LIN {X 0,Y 190.338,Z 370.744,A -85,B 0,C 180,E1 -22072.2,E2 -22072.2} C_VEL
LIN {X 0,Y 193.251,Z 362.35,A -85,B 0,C 180,E1 -22075.296,E2 -22075.296} C_VEL
LIN {X 0,Y 196.197,Z 353.832,A -85,B 0,C 180,E1 -22077.752,E2 -22077.752} C_VEL
LIN {X 0,Y 199.587,Z 343.318,A -85,B 0,C 180,E1 -22080.116,E2 -22080.116} C_VEL
LIN {X 0,Y 202.903,Z 331.483,A -85,B 0,C 180,E1 -22082.176,E2 -22082.176} C_VEL
LIN {X 0,Y 205.757,Z 319.558,A -85,B 0,C 180,E1 -22083.712,E2 -22083.712} C_VEL
LIN {X 0,Y 208.119,Z 307.146,A -85,B 0,C 180,E1 -22084.886,E2 -22084.886} C_VEL
LIN {X 0,Y 209.878,Z 294.163,A -85,B 0,C 180,E1 -22085.737,E2 -22085.737} C_VEL
LIN {X 0,Y 210.855,Z 279.203,A -85,B 0,C 180,E1 -22086.333,E2 -22086.333} C_VEL
LIN {X 0,Y 212.644,Z 242.014,A -85,B 0,C 180,E1 -22087.513,E2 -22087.513} C_VEL
LIN {X 0,Y 211,Z 228.178,A -85,B 0,C 180,E1 -22088.437,E2 -22088.437} C_VEL
LIN {X 0,Y 205.351,Z 214.211,A -85,B 0,C 180,E1 -22090.309,E2 -22090.309} C_VEL
LIN {X 0,Y 199.119,Z 201.239,A -85,B 0,C 180,E1 -22092.447,E2 -22092.447} C_VEL
LIN {X 0,Y 194.454,Z 192.885,A -85,B 0,C 180,E1 -22094.123,E2 -22094.123} C_VEL
LIN {X 0,Y 191.867,Z 188.463,A -85,B 0,C 180,E1 -22095.097,E2 -22095.097} C_VEL
LIN {X 0,Y 189.584,Z 184.486,A -85,B 0,C 180,E1 -22095.998,E2 -22095.998} C_VEL
LIN {X 0,Y 186.826,Z 180.02,A -85,B 0,C 180,E1 -22097.117,E2 -22097.117} C_VEL
LIN {X 0,Y 186.602,Z 179.438,A -85,B 0,C 180,E1 -22097.318,E2 -22097.318} C_VEL
LIN {X 0,Y 185.459,Z 175.379,A -85,B 0,C 180,E1 -22100.247,E2 -22100.247} C_VEL
LIN {X 0,Y 185.496,Z 175.37,A -85,B 0,C 180,E1 -22102.713,E2 -22102.713} C_VEL
LIN {X 0,Y 185.525,Z 175.365,A -85,B 0,C 180,E1 -22107.971,E2 -22107.971} C_VEL
LIN {X 0,Y 185.542,Z 175.361,A -85,B 0,C 180,E1 -22110.595,E2 -22110.595} C_VEL
LIN {X 0,Y 185.557,Z 175.366,A -85,B 0,C 180,E1 -22115.378,E2 -22115.378} C_VEL
LIN {X 0,Y 185.619,Z 175.361,A -85,B 0,C 180,E1 -22121.178,E2 -22121.178} C_VEL
LIN {X 0,Y 185.691,Z 175.355,A -85,B 0,C 180,E1 -22126.874,E2 -22126.874} C_VEL
LIN {X 0,Y 185.962,Z 175.306,A -85,B 0,C 180,E1 -22131.305,E2 -22131.305} C_VEL
LIN {X 0,Y 186.164,Z 175.274,A -85,B 0,C 180,E1 -22137.837,E2 -22137.837} C_VEL
LIN {X 0,Y 186.371,Z 175.265,A -85,B 0,C 180,E1 -22140,E2 -22140} C_VEL
LIN {X 0,Y 185.875,Z 175.31,A -85,B 0,C 180,E1 -22144.337,E2 -22144.337} C_VEL
LIN {X 0,Y 185.968,Z 175.32,A -85,B 0,C 180,E1 -22148.695,E2 -22148.695} C_VEL
LIN {X 0,Y 185.679,Z 175.336,A -85,B 0,C 180,E1 -22153.127,E2 -22153.127} C_VEL
LIN {X 0,Y 185.619,Z 175.347,A -85,B 0,C 180,E1 -22158.822,E2 -22158.822} C_VEL
LIN {X 0,Y 185.572,Z 175.359,A -85,B 0,C 180,E1 -22164.647,E2 -22164.647} C_VEL
LIN {X 0,Y 185.539,Z 175.372,A -85,B 0,C 180,E1 -22169.5,E2 -22169.5} C_VEL
LIN {X 0,Y 185.492,Z 175.38,A -85,B 0,C 180,E1 -22174.634,E2 -22174.634} C_VEL
LIN {X 0,Y 185.495,Z 175.377,A -85,B 0,C 180,E1 -22177.316,E2 -22177.316} C_VEL
LIN {X 0,Y 185.432,Z 175.385,A -85,B 0,C 180,E1 -22182.703,E2 -22182.703} C_VEL
LIN {X 0,Y 186.407,Z 178.185,A -85,B 0,C 180,E1 -22183.202,E2 -22183.202} C_VEL
LIN {X 0,Y 188.839,Z 180.945,A -85,B 0,C 180,E1 -22184.138,E2 -22184.138} C_VEL
LIN {X 0,Y 191.097,Z 184.353,A -85,B 0,C 180,E1 -22185.017,E2 -22185.017} C_VEL
LIN {X 0,Y 197.59,Z 193.93,A -85,B 0,C 180,E1 -22187.354,E2 -22187.354} C_VEL
LIN {X 0,Y 204.857,Z 205.887,A -85,B 0,C 180,E1 -22189.759,E2 -22189.759} C_VEL
LIN {X 0,Y 209.367,Z 214.642,A -85,B 0,C 180,E1 -22191.186,E2 -22191.186} C_VEL
LIN {X 0,Y 213.513,Z 224.523,A -85,B 0,C 180,E1 -22192.497,E2 -22192.497} C_VEL
LIN {X 0,Y 210.927,Z 276.622,A -85,B 0,C 180,E1 -22194.185,E2 -22194.185} C_VEL
LIN {X 0,Y 209.573,Z 289.686,A -85,B 0,C 180,E1 -22194.928,E2 -22194.928} C_VEL
LIN {X 0,Y 207.599,Z 302.646,A -85,B 0,C 180,E1 -22196.044,E2 -22196.044} C_VEL
LIN {X 0,Y 205.428,Z 313.931,A -85,B 0,C 180,E1 -22197.398,E2 -22197.398} C_VEL
LIN {X 0,Y 202.486,Z 325.552,A -85,B 0,C 180,E1 -22199.208,E2 -22199.208} C_VEL
LIN {X 0,Y 199.477,Z 335.985,A -85,B 0,C 180,E1 -22201.314,E2 -22201.314} C_VEL
LIN {X 0,Y 196.603,Z 345.342,A -85,B 0,C 180,E1 -22203.736,E2 -22203.736} C_VEL
LIN {X 0,Y 193.541,Z 353.735,A -85,B 0,C 180,E1 -22206.458,E2 -22206.458} C_VEL
LIN {X 0,Y 190.64,Z 361.13,A -85,B 0,C 180,E1 -22209.501,E2 -22209.501} C_VEL
LIN {X 0,Y 188.279,Z 367.06,A -85,B 0,C 180,E1 -22212.627,E2 -22212.627} C_VEL
LIN {X 0,Y 186.38,Z 371.743,A -85,B 0,C 180,E1 -22215.814,E2 -22215.814} C_VEL
LIN {X 0,Y 184.952,Z 375.324,A -85,B 0,C 180,E1 -22219.049,E2 -22219.049} C_VEL
LIN {X 0,Y 184.328,Z 377.17,A -85,B 0,C 180,E1 -22221.229,E2 -22221.229} C_VEL
LIN {X 0,Y 183.778,Z 378.789,A -85,B 0,C 180,E1 -22223.877,E2 -22223.877} C_VEL
LIN {X 0,Y 183.373,Z 380.147,A -85,B 0,C 180,E1 -22227.805,E2 -22227.805} C_VEL
LIN {X 0,Y 183.339,Z 380.373,A -85,B 0,C 180,E1 -22230.001,E2 -22230.001} C_VEL
LIN {X 0,Y 183.372,Z 380.18,A -85,B 0,C 180,E1 -22232.198,E2 -22232.198} C_VEL
LIN {X 0,Y 183.856,Z 378.631,A -85,B 0,C 180,E1 -22236.586,E2 -22236.586} C_VEL
LIN {X 0,Y 184.327,Z 377.277,A -85,B 0,C 180,E1 -22238.774,E2 -22238.774} C_VEL
LIN {X 0,Y 185.352,Z 374.417,A -85,B 0,C 180,E1 -22242.038,E2 -22242.038} C_VEL
LIN {X 0,Y 186.915,Z 370.531,A -85,B 0,C 180,E1 -22245.261,E2 -22245.261} C_VEL
LIN {X 0,Y 188.992,Z 365.515,A -85,B 0,C 180,E1 -22248.427,E2 -22248.427} C_VEL
LIN {X 0,Y 191.478,Z 359.197,A -85,B 0,C 180,E1 -22251.534,E2 -22251.534} C_VEL
LIN {X 0,Y 194.571,Z 351.285,A -85,B 0,C 180,E1 -22254.544,E2 -22254.544} C_VEL
LIN {X 0,Y 197.641,Z 342.318,A -85,B 0,C 180,E1 -22257.253,E2 -22257.253} C_VEL
LIN {X 0,Y 200.702,Z 332.281,A -85,B 0,C 180,E1 -22259.645,E2 -22259.645} C_VEL
LIN {X 0,Y 203.852,Z 320.867,A -85,B 0,C 180,E1 -22261.72,E2 -22261.72} C_VEL
LIN {X 0,Y 206.468,Z 309.65,A -85,B 0,C 180,E1 -22263.291,E2 -22263.291} C_VEL
LIN {X 0,Y 208.567,Z 298.245,A -85,B 0,C 180,E1 -22264.509,E2 -22264.509} C_VEL
LIN {X 0,Y 210.229,Z 285.423,A -85,B 0,C 180,E1 -22265.49,E2 -22265.49} C_VEL
LIN {X 0,Y 211.371,Z 272.725,A -85,B 0,C 180,E1 -22266.089,E2 -22266.089} C_VEL
LIN {X 0,Y 213.621,Z 224.617,A -85,B 0,C 180,E1 -22267.642,E2 -22267.642} C_VEL
LIN {X 0,Y 208.154,Z 211.914,A -85,B 0,C 180,E1 -22269.377,E2 -22269.377} C_VEL
LIN {X 0,Y 201.122,Z 199.457,A -85,B 0,C 180,E1 -22271.638,E2 -22271.638} C_VEL
LIN {X 0,Y 194.074,Z 188.613,A -85,B 0,C 180,E1 -22274.078,E2 -22274.078} C_VEL
LIN {X 0,Y 190.919,Z 184.144,A -85,B 0,C 180,E1 -22275.244,E2 -22275.244} C_VEL
LIN {X 0,Y 188.768,Z 180.719,A -85,B 0,C 180,E1 -22276.096,E2 -22276.096} C_VEL
LIN {X 0,Y 186.303,Z 178.004,A -85,B 0,C 180,E1 -22277.047,E2 -22277.047} C_VEL
LIN {X 0,Y 185.436,Z 175.386,A -85,B 0,C 180,E1 -22277.533,E2 -22277.533} C_VEL
LIN {X 0,Y 185.502,Z 175.376,A -85,B 0,C 180,E1 -22282.714,E2 -22282.714} C_VEL
LIN {X 0,Y 185.532,Z 175.374,A -85,B 0,C 180,E1 -22287.972,E2 -22287.972} C_VEL
LIN {X 0,Y 185.549,Z 175.354,A -85,B 0,C 180,E1 -22290.595,E2 -22290.595} C_VEL
LIN {X 0,Y 185.582,Z 175.362,A -85,B 0,C 180,E1 -22295.382,E2 -22295.382} C_VEL
LIN {X 0,Y 185.627,Z 175.363,A -85,B 0,C 180,E1 -22301.178,E2 -22301.178} C_VEL
LIN {X 0,Y 185.701,Z 175.341,A -85,B 0,C 180,E1 -22306.875,E2 -22306.875} C_VEL
LIN {X 0,Y 185.974,Z 175.303,A -85,B 0,C 180,E1 -22311.306,E2 -22311.306} C_VEL
LIN {X 0,Y 186.175,Z 175.293,A -85,B 0,C 180,E1 -22317.836,E2 -22317.836} C_VEL
LIN {X 0,Y 186.379,Z 175.247,A -85,B 0,C 180,E1 -22320,E2 -22320} C_VEL
LIN {X 0,Y 185.876,Z 175.328,A -85,B 0,C 180,E1 -22324.337,E2 -22324.337} C_VEL
LIN {X 0,Y 185.97,Z 175.296,A -85,B 0,C 180,E1 -22328.694,E2 -22328.694} C_VEL
LIN {X 0,Y 185.683,Z 175.354,A -85,B 0,C 180,E1 -22333.126,E2 -22333.126} C_VEL
LIN {X 0,Y 185.626,Z 175.355,A -85,B 0,C 180,E1 -22338.821,E2 -22338.821} C_VEL
LIN {X 0,Y 185.545,Z 175.362,A -85,B 0,C 180,E1 -22344.623,E2 -22344.623} C_VEL
LIN {X 0,Y 185.545,Z 175.36,A -85,B 0,C 180,E1 -22349.499,E2 -22349.499} C_VEL
LIN {X 0,Y 185.498,Z 175.368,A -85,B 0,C 180,E1 -22354.632,E2 -22354.632} C_VEL
LIN {X 0,Y 185.484,Z 175.38,A -85,B 0,C 180,E1 -22359.659,E2 -22359.659} C_VEL
LIN {X 0,Y 186.761,Z 179.671,A -85,B 0,C 180,E1 -22362.728,E2 -22362.728} C_VEL
LIN {X 0,Y 189.367,Z 184.168,A -85,B 0,C 180,E1 -22363.809,E2 -22363.809} C_VEL
LIN {X 0,Y 190.744,Z 186.397,A -85,B 0,C 180,E1 -22364.352,E2 -22364.352} C_VEL
LIN {X 0,Y 196.414,Z 196.178,A -85,B 0,C 180,E1 -22366.49,E2 -22366.49} C_VEL
LIN {X 0,Y 201.168,Z 205.286,A -85,B 0,C 180,E1 -22368.178,E2 -22368.178} C_VEL
LIN {X 0,Y 206.364,Z 216.482,A -85,B 0,C 180,E1 -22369.945,E2 -22369.945} C_VEL
LIN {X 0,Y 211.188,Z 228.61,A -85,B 0,C 180,E1 -22371.544,E2 -22371.544} C_VEL
LIN {X 0,Y 212.771,Z 242.115,A -85,B 0,C 180,E1 -22372.443,E2 -22372.443} C_VEL
LIN {X 0,Y 211.518,Z 269.834,A -85,B 0,C 180,E1 -22373.338,E2 -22373.338} C_VEL
LIN {X 0,Y 210.655,Z 275.689,A -85,B 0,C 180,E1 -22373.4,E2 -22373.4} C_VEL
LIN {X 0,Y 205.321,Z 292.719,A -85,B 0,C 180,E1 -22373.17,E2 -22373.17} C_VEL
LIN {X 0,Y 203.85,Z 298.411,A -85,B 0,C 180,E1 -22373.322,E2 -22373.322} C_VEL
LIN {X 0,Y 203.519,Z 300.309,A -85,B 0,C 180,E1 -22373.435,E2 -22373.435} C_VEL
LIN {X 0,Y 201.23,Z 313.562,A -85,B 0,C 180,E1 -22374.504,E2 -22374.504} C_VEL
LIN {X 0,Y 198.611,Z 325.214,A -85,B 0,C 180,E1 -22375.823,E2 -22375.823} C_VEL
LIN {X 0,Y 195.366,Z 337.148,A -85,B 0,C 180,E1 -22377.648,E2 -22377.648} C_VEL
LIN {X 0,Y 192.03,Z 347.789,A -85,B 0,C 180,E1 -22379.785,E2 -22379.785} C_VEL
LIN {X 0,Y 188.635,Z 357.381,A -85,B 0,C 180,E1 -22382.243,E2 -22382.243} C_VEL
LIN {X 0,Y 185.76,Z 365.251,A -85,B 0,C 180,E1 -22384.809,E2 -22384.809} C_VEL
LIN {X 0,Y 182.859,Z 372.945,A -85,B 0,C 180,E1 -22387.991,E2 -22387.991} C_VEL
LIN {X 0,Y 180.732,Z 378.219,A -85,B 0,C 180,E1 -22390.698,E2 -22390.698} C_VEL
LIN {X 0,Y 178.6,Z 383.328,A -85,B 0,C 180,E1 -22394.01,E2 -22394.01} C_VEL
LIN {X 0,Y 177.263,Z 387.31,A -85,B 0,C 180,E1 -22397.404,E2 -22397.404} C_VEL
LIN {X 0,Y 176.398,Z 390.256,A -85,B 0,C 180,E1 -22400.829,E2 -22400.829} C_VEL
LIN {X 0,Y 175.973,Z 392.666,A -85,B 0,C 180,E1 -22405.417,E2 -22405.417} C_VEL
LIN {X 0,Y 176.02,Z 393.282,A -85,B 0,C 180,E1 -22407.711,E2 -22407.711} C_VEL
LIN {X 0,Y 176.171,Z 393.501,A -85,B 0,C 180,E1 -22409.999,E2 -22409.999} C_VEL
LIN {X 0,Y 175.995,Z 393.047,A -85,B 0,C 180,E1 -22413.318,E2 -22413.318} C_VEL
LIN {X 0,Y 176.115,Z 391.631,A -85,B 0,C 180,E1 -22416.874,E2 -22416.874} C_VEL
LIN {X 0,Y 176.41,Z 390.213,A -85,B 0,C 180,E1 -22419.168,E2 -22419.168} C_VEL
LIN {X 0,Y 177.264,Z 387.248,A -85,B 0,C 180,E1 -22422.594,E2 -22422.594} C_VEL
LIN {X 0,Y 178.598,Z 383.242,A -85,B 0,C 180,E1 -22425.988,E2 -22425.988} C_VEL
LIN {X 0,Y 181.048,Z 377.099,A -85,B 0,C 180,E1 -22429.855,E2 -22429.855} C_VEL
LIN {X 0,Y 183.924,Z 369.91,A -85,B 0,C 180,E1 -22433.291,E2 -22433.291} C_VEL
LIN {X 0,Y 186.823,Z 362.087,A -85,B 0,C 180,E1 -22436.231,E2 -22436.231} C_VEL
LIN {X 0,Y 189.932,Z 353.57,A -85,B 0,C 180,E1 -22438.751,E2 -22438.751} C_VEL
LIN {X 0,Y 193.478,Z 343.055,A -85,B 0,C 180,E1 -22441.171,E2 -22441.171} C_VEL
LIN {X 0,Y 196.927,Z 331.219,A -85,B 0,C 180,E1 -22443.277,E2 -22443.277} C_VEL
LIN {X 0,Y 199.897,Z 319.293,A -85,B 0,C 180,E1 -22444.84,E2 -22444.84} C_VEL
LIN {X 0,Y 202.347,Z 306.879,A -85,B 0,C 180,E1 -22446.033,E2 -22446.033} C_VEL
LIN {X 0,Y 204.161,Z 293.861,A -85,B 0,C 180,E1 -22446.902,E2 -22446.902} C_VEL
LIN {X 0,Y 205.185,Z 278.413,A -85,B 0,C 180,E1 -22447.528,E2 -22447.528} C_VEL
LIN {X 0,Y 207.013,Z 243.038,A -85,B 0,C 180,E1 -22448.662,E2 -22448.662} C_VEL
LIN {X 0,Y 205.469,Z 230.374,A -85,B 0,C 180,E1 -22449.562,E2 -22449.562} C_VEL
LIN {X 0,Y 199.683,Z 216.169,A -85,B 0,C 180,E1 -22451.597,E2 -22451.597} C_VEL
LIN {X 0,Y 193.673,Z 203.584,A -85,B 0,C 180,E1 -22453.807,E2 -22453.807} C_VEL
LIN {X 0,Y 187.565,Z 192.871,A -85,B 0,C 180,E1 -22456.18,E2 -22456.18} C_VEL
LIN {X 0,Y 185.154,Z 188.806,A -85,B 0,C 180,E1 -22457.181,E2 -22457.181} C_VEL
LIN {X 0,Y 182.179,Z 184.022,A -85,B 0,C 180,E1 -22458.467,E2 -22458.467} C_VEL
LIN {X 0,Y 179.412,Z 179.562,A -85,B 0,C 180,E1 -22459.733,E2 -22459.733} C_VEL
LIN {X 0,Y 179.064,Z 178.458,A -85,B 0,C 180,E1 -22460.373,E2 -22460.373} C_VEL
LIN {X 0,Y 178.46,Z 176.248,A -85,B 0,C 180,E1 -22462.161,E2 -22462.161} C_VEL
LIN {X 0,Y 178.478,Z 176.241,A -85,B 0,C 180,E1 -22466.545,E2 -22466.545} C_VEL
LIN {X 0,Y 178.434,Z 176.241,A -85,B 0,C 180,E1 -22471.794,E2 -22471.794} C_VEL
LIN {X 0,Y 178.499,Z 176.247,A -85,B 0,C 180,E1 -22474.896,E2 -22474.896} C_VEL
LIN {X 0,Y 178.596,Z 176.23,A -85,B 0,C 180,E1 -22481.651,E2 -22481.651} C_VEL
LIN {X 0,Y 178.617,Z 176.236,A -85,B 0,C 180,E1 -22486.345,E2 -22486.345} C_VEL
LIN {X 0,Y 178.894,Z 176.183,A -85,B 0,C 180,E1 -22490.959,E2 -22490.959} C_VEL
LIN {X 0,Y 179.112,Z 176.152,A -85,B 0,C 180,E1 -22497.751,E2 -22497.751} C_VEL
LIN {X 0,Y 179.337,Z 176.141,A -85,B 0,C 180,E1 -22500,E2 -22500} C_VEL
LIN {X 0,Y 178.824,Z 176.187,A -85,B 0,C 180,E1 -22504.508,E2 -22504.508} C_VEL
LIN {X 0,Y 178.899,Z 176.201,A -85,B 0,C 180,E1 -22509.041,E2 -22509.041} C_VEL
LIN {X 0,Y 178.611,Z 176.219,A -85,B 0,C 180,E1 -22513.656,E2 -22513.656} C_VEL
LIN {X 0,Y 178.548,Z 176.225,A -85,B 0,C 180,E1 -22519.152,E2 -22519.152} C_VEL
LIN {X 0,Y 178.51,Z 176.234,A -85,B 0,C 180,E1 -22525.112,E2 -22525.112} C_VEL
LIN {X 0,Y 178.455,Z 176.244,A -85,B 0,C 180,E1 -22530.796,E2 -22530.796} C_VEL
LIN {X 0,Y 178.478,Z 176.254,A -85,B 0,C 180,E1 -22534.219,E2 -22534.219} C_VEL
LIN {X 0,Y 178.43,Z 176.313,A -85,B 0,C 180,E1 -22540.257,E2 -22540.257} C_VEL
LIN {X 0,Y 179.241,Z 178.811,A -85,B 0,C 180,E1 -22540.716,E2 -22540.716} C_VEL
LIN {X 0,Y 181.274,Z 181.131,A -85,B 0,C 180,E1 -22541.601,E2 -22541.601} C_VEL
LIN {X 0,Y 182.051,Z 182.176,A -85,B 0,C 180,E1 -22541.939,E2 -22541.939} C_VEL
LIN {X 0,Y 184.266,Z 185.378,A -85,B 0,C 180,E1 -22542.889,E2 -22542.889} C_VEL
LIN {X 0,Y 185.733,Z 187.418,A -85,B 0,C 180,E1 -22543.491,E2 -22543.491} C_VEL
LIN {X 0,Y 191.573,Z 195.936,A -85,B 0,C 180,E1 -22545.76,E2 -22545.76} C_VEL
LIN {X 0,Y 198.102,Z 206.422,A -85,B 0,C 180,E1 -22548.093,E2 -22548.093} C_VEL
LIN {X 0,Y 203.953,Z 217.315,A -85,B 0,C 180,E1 -22550.06,E2 -22550.06} C_VEL
LIN {X 0,Y 207.857,Z 226.554,A -85,B 0,C 180,E1 -22551.367,E2 -22551.367} C_VEL
LIN {X 0,Y 205.217,Z 277.095,A -85,B 0,C 180,E1 -22553.039,E2 -22553.039} C_VEL
LIN {X 0,Y 203.795,Z 290.112,A -85,B 0,C 180,E1 -22553.796,E2 -22553.796} C_VEL
LIN {X 0,Y 201.77,Z 302.912,A -85,B 0,C 180,E1 -22554.922,E2 -22554.922} C_VEL
LIN {X 0,Y 199.509,Z 314.194,A -85,B 0,C 180,E1 -22556.304,E2 -22556.304} C_VEL
LIN {X 0,Y 196.433,Z 325.815,A -85,B 0,C 180,E1 -22558.15,E2 -22558.15} C_VEL
LIN {X 0,Y 193.278,Z 336.247,A -85,B 0,C 180,E1 -22560.303,E2 -22560.303} C_VEL
LIN {X 0,Y 190.18,Z 345.847,A -85,B 0,C 180,E1 -22562.865,E2 -22562.865} C_VEL
LIN {X 0,Y 187.065,Z 353.996,A -85,B 0,C 180,E1 -22565.591,E2 -22565.591} C_VEL
LIN {X 0,Y 184.009,Z 361.391,A -85,B 0,C 180,E1 -22568.727,E2 -22568.727} C_VEL
LIN {X 0,Y 181.529,Z 367.32,A -85,B 0,C 180,E1 -22571.959,E2 -22571.959} C_VEL
LIN {X 0,Y 179.509,Z 372.004,A -85,B 0,C 180,E1 -22575.259,E2 -22575.259} C_VEL
LIN {X 0,Y 178.004,Z 375.584,A -85,B 0,C 180,E1 -22578.616,E2 -22578.616} C_VEL
LIN {X 0,Y 177.308,Z 377.43,A -85,B 0,C 180,E1 -22580.879,E2 -22580.879} C_VEL
LIN {X 0,Y 176.658,Z 379.245,A -85,B 0,C 180,E1 -22584.035,E2 -22584.035} C_VEL
LIN {X 0,Y 176.283,Z 380.406,A -85,B 0,C 180,E1 -22587.716,E2 -22587.716} C_VEL
LIN {X 0,Y 176.244,Z 380.632,A -85,B 0,C 180,E1 -22590.001,E2 -22590.001} C_VEL
LIN {X 0,Y 176.283,Z 380.439,A -85,B 0,C 180,E1 -22592.286,E2 -22592.286} C_VEL
LIN {X 0,Y 176.813,Z 378.889,A -85,B 0,C 180,E1 -22596.85,E2 -22596.85} C_VEL
LIN {X 0,Y 177.307,Z 377.536,A -85,B 0,C 180,E1 -22599.124,E2 -22599.124} C_VEL
LIN {X 0,Y 178.406,Z 374.676,A -85,B 0,C 180,E1 -22602.514,E2 -22602.514} C_VEL
LIN {X 0,Y 180.081,Z 370.789,A -85,B 0,C 180,E1 -22605.855,E2 -22605.855} C_VEL
LIN {X 0,Y 182.249,Z 365.774,A -85,B 0,C 180,E1 -22609.135,E2 -22609.135} C_VEL
LIN {X 0,Y 184.912,Z 359.454,A -85,B 0,C 180,E1 -22612.339,E2 -22612.339} C_VEL
LIN {X 0,Y 188.146,Z 351.541,A -85,B 0,C 180,E1 -22615.441,E2 -22615.441} C_VEL
LIN {X 0,Y 191.149,Z 343.155,A -85,B 0,C 180,E1 -22618.065,E2 -22618.065} C_VEL
LIN {X 0,Y 194.204,Z 333.638,A -85,B 0,C 180,E1 -22620.441,E2 -22620.441} C_VEL
LIN {X 0,Y 197.488,Z 322.542,A -85,B 0,C 180,E1 -22622.565,E2 -22622.565} C_VEL
LIN {X 0,Y 200.178,Z 311.664,A -85,B 0,C 180,E1 -22624.177,E2 -22624.177} C_VEL
LIN {X 0,Y 202.535,Z 299.636,A -85,B 0,C 180,E1 -22625.538,E2 -22625.538} C_VEL
LIN {X 0,Y 204.383,Z 286.815,A -85,B 0,C 180,E1 -22626.571,E2 -22626.571} C_VEL
LIN {X 0,Y 205.688,Z 273.109,A -85,B 0,C 180,E1 -22627.244,E2 -22627.244} C_VEL
LIN {X 0,Y 207.96,Z 226.677,A -85,B 0,C 180,E1 -22628.775,E2 -22628.775} C_VEL
LIN {X 0,Y 203.224,Z 215.624,A -85,B 0,C 180,E1 -22630.367,E2 -22630.367} C_VEL
LIN {X 0,Y 196.493,Z 203.667,A -85,B 0,C 180,E1 -22632.653,E2 -22632.653} C_VEL
LIN {X 0,Y 189.998,Z 193.528,A -85,B 0,C 180,E1 -22635.031,E2 -22635.031} C_VEL
LIN {X 0,Y 184.57,Z 185.682,A -85,B 0,C 180,E1 -22637.199,E2 -22637.199} C_VEL
LIN {X 0,Y 182.212,Z 182.471,A -85,B 0,C 180,E1 -22638.199,E2 -22638.199} C_VEL
LIN {X 0,Y 181.59,Z 181.34,A -85,B 0,C 180,E1 -22638.487,E2 -22638.487} C_VEL
LIN {X 0,Y 179.399,Z 179.068,A -85,B 0,C 180,E1 -22639.428,E2 -22639.428} C_VEL
LIN {X 0,Y 178.421,Z 176.245,A -85,B 0,C 180,E1 -22640.017,E2 -22640.017} C_VEL
LIN {X 0,Y 178.484,Z 176.238,A -85,B 0,C 180,E1 -22645.782,E2 -22645.782} C_VEL
LIN {X 0,Y 178.483,Z 176.236,A -85,B 0,C 180,E1 -22650.03,E2 -22650.03} C_VEL
LIN {X 0,Y 178.517,Z 176.245,A -85,B 0,C 180,E1 -22654.889,E2 -22654.889} C_VEL
LIN {X 0,Y 178.608,Z 176.236,A -85,B 0,C 180,E1 -22661.652,E2 -22661.652} C_VEL
LIN {X 0,Y 178.628,Z 176.215,A -85,B 0,C 180,E1 -22666.345,E2 -22666.345} C_VEL
LIN {X 0,Y 178.905,Z 176.186,A -85,B 0,C 180,E1 -22670.959,E2 -22670.959} C_VEL
LIN {X 0,Y 179.123,Z 176.172,A -85,B 0,C 180,E1 -22677.751,E2 -22677.751} C_VEL
LIN {X 0,Y 179.344,Z 176.122,A -85,B 0,C 180,E1 -22680,E2 -22680} C_VEL
LIN {X 0,Y 178.825,Z 176.208,A -85,B 0,C 180,E1 -22684.508,E2 -22684.508} C_VEL
LIN {X 0,Y 178.901,Z 176.174,A -85,B 0,C 180,E1 -22689.041,E2 -22689.041} C_VEL
LIN {X 0,Y 178.613,Z 176.234,A -85,B 0,C 180,E1 -22693.656,E2 -22693.656} C_VEL
LIN {X 0,Y 178.555,Z 176.239,A -85,B 0,C 180,E1 -22699.151,E2 -22699.151} C_VEL
LIN {X 0,Y 178.466,Z 176.247,A -85,B 0,C 180,E1 -22705.076,E2 -22705.076} C_VEL
LIN {X 0,Y 178.461,Z 176.252,A -85,B 0,C 180,E1 -22710.794,E2 -22710.794} C_VEL
LIN {X 0,Y 178.483,Z 176.24,A -85,B 0,C 180,E1 -22714.218,E2 -22714.218} C_VEL
LIN {X 0,Y 178.466,Z 176.303,A -85,B 0,C 180,E1 -22717.837,E2 -22717.837} C_VEL
LIN {X 0,Y 179.343,Z 179.382,A -85,B 0,C 180,E1 -22720.101,E2 -22720.101} C_VEL
LIN {X 0,Y 181.706,Z 183.34,A -85,B 0,C 180,E1 -22721.203,E2 -22721.203} C_VEL
LIN {X 0,Y 183.511,Z 186.016,A -85,B 0,C 180,E1 -22721.991,E2 -22721.991} C_VEL
LIN {X 0,Y 187.016,Z 191.797,A -85,B 0,C 180,E1 -22723.476,E2 -22723.476} C_VEL
LIN {X 0,Y 192.602,Z 201.679,A -85,B 0,C 180,E1 -22725.692,E2 -22725.692} C_VEL
LIN {X 0,Y 198.038,Z 212.402,A -85,B 0,C 180,E1 -22727.711,E2 -22727.711} C_VEL
LIN {X 0,Y 203.968,Z 226.256,A -85,B 0,C 180,E1 -22729.823,E2 -22729.823} C_VEL
LIN {X 0,Y 205.855,Z 231.451,A -85,B 0,C 180,E1 -22730.491,E2 -22730.491} C_VEL
LIN {X 0,Y 207.131,Z 244.58,A -85,B 0,C 180,E1 -22731.35,E2 -22731.35} C_VEL
LIN {X 0,Y 204.767,Z 289.08,A -85,B 0,C 180,E1 -22732.823,E2 -22732.823} C_VEL
LIN {X 0,Y 203.519,Z 300.309,A -85,B 0,C 180,E1 -22733.435,E2 -22733.435} C_VEL
LIN {X 0,Y 202.627,Z 304.081,A -85,B 0,C 180,E1 -22733.631,E2 -22733.631} C_VEL
LIN {X 0,Y 199.697,Z 311.381,A -85,B 0,C 180,E1 -22733.902,E2 -22733.902} C_VEL
LIN {X 0,Y 196.103,Z 318.417,A -85,B 0,C 180,E1 -22734.185,E2 -22734.185} C_VEL
LIN {X 0,Y 192.888,Z 325.441,A -85,B 0,C 180,E1 -22734.746,E2 -22734.746} C_VEL
LIN {X 0,Y 191.747,Z 328.837,A -85,B 0,C 180,E1 -22735.187,E2 -22735.187} C_VEL
LIN {X 0,Y 188.619,Z 339.483,A -85,B 0,C 180,E1 -22736.979,E2 -22736.979} C_VEL
LIN {X 0,Y 185.153,Z 349.638,A -85,B 0,C 180,E1 -22739.173,E2 -22739.173} C_VEL
LIN {X 0,Y 181.712,Z 358.795,A -85,B 0,C 180,E1 -22741.719,E2 -22741.719} C_VEL
LIN {X 0,Y 178.317,Z 367.44,A -85,B 0,C 180,E1 -22744.799,E2 -22744.799} C_VEL
LIN {X 0,Y 175.277,Z 374.924,A -85,B 0,C 180,E1 -22748.228,E2 -22748.228} C_VEL
LIN {X 0,Y 172.462,Z 381.478,A -85,B 0,C 180,E1 -22752.203,E2 -22752.203} C_VEL
LIN {X 0,Y 170.694,Z 385.821,A -85,B 0,C 180,E1 -22755.697,E2 -22755.697} C_VEL
LIN {X 0,Y 169.961,Z 388.129,A -85,B 0,C 180,E1 -22758.067,E2 -22758.067} C_VEL
LIN {X 0,Y 169.364,Z 389.997,A -85,B 0,C 180,E1 -22760.444,E2 -22760.444} C_VEL
LIN {X 0,Y 168.875,Z 392.406,A -85,B 0,C 180,E1 -22765.224,E2 -22765.224} C_VEL
LIN {X 0,Y 168.947,Z 393.024,A -85,B 0,C 180,E1 -22767.615,E2 -22767.615} C_VEL
LIN {X 0,Y 169.075,Z 393.242,A -85,B 0,C 180,E1 -22769.999,E2 -22769.999} C_VEL
LIN {X 0,Y 168.91,Z 392.873,A -85,B 0,C 180,E1 -22773.041,E2 -22773.041} C_VEL
LIN {X 0,Y 169.036,Z 391.371,A -85,B 0,C 180,E1 -22777.164,E2 -22777.164} C_VEL
LIN {X 0,Y 169.374,Z 389.952,A -85,B 0,C 180,E1 -22779.553,E2 -22779.553} C_VEL
LIN {X 0,Y 170.294,Z 386.986,A -85,B 0,C 180,E1 -22783.118,E2 -22783.118} C_VEL
LIN {X 0,Y 171.766,Z 382.981,A -85,B 0,C 180,E1 -22786.642,E2 -22786.642} C_VEL
LIN {X 0,Y 174.339,Z 376.837,A -85,B 0,C 180,E1 -22790.653,E2 -22790.653} C_VEL
LIN {X 0,Y 177.15,Z 370.236,A -85,B 0,C 180,E1 -22793.942,E2 -22793.942} C_VEL
LIN {X 0,Y 180.452,Z 361.824,A -85,B 0,C 180,E1 -22797.232,E2 -22797.232} C_VEL
LIN {X 0,Y 183.724,Z 353.307,A -85,B 0,C 180,E1 -22799.819,E2 -22799.819} C_VEL
LIN {X 0,Y 187.433,Z 342.792,A -85,B 0,C 180,E1 -22802.296,E2 -22802.296} C_VEL
LIN {X 0,Y 190.613,Z 332.387,A -85,B 0,C 180,E1 -22804.211,E2 -22804.211} C_VEL
LIN {X 0,Y 193.669,Z 320.976,A -85,B 0,C 180,E1 -22805.812,E2 -22805.812} C_VEL
LIN {X 0,Y 196.21,Z 309.217,A -85,B 0,C 180,E1 -22807.026,E2 -22807.026} C_VEL
LIN {X 0,Y 198.213,Z 296.275,A -85,B 0,C 180,E1 -22807.972,E2 -22807.972} C_VEL
LIN {X 0,Y 199.355,Z 283.414,A -85,B 0,C 180,E1 -22808.583,E2 -22808.583} C_VEL
LIN {X 0,Y 201.404,Z 243.599,A -85,B 0,C 180,E1 -22809.912,E2 -22809.912} C_VEL
LIN {X 0,Y 200.12,Z 232.927,A -85,B 0,C 180,E1 -22810.708,E2 -22810.708} C_VEL
LIN {X 0,Y 194.41,Z 218.79,A -85,B 0,C 180,E1 -22812.849,E2 -22812.849} C_VEL
LIN {X 0,Y 189.012,Z 207.503,A -85,B 0,C 180,E1 -22814.959,E2 -22814.959} C_VEL
LIN {X 0,Y 182.035,Z 194.852,A -85,B 0,C 180,E1 -22817.893,E2 -22817.893} C_VEL
LIN {X 0,Y 178.003,Z 188.501,A -85,B 0,C 180,E1 -22819.72,E2 -22819.72} C_VEL
LIN {X 0,Y 175.015,Z 183.777,A -85,B 0,C 180,E1 -22821.177,E2 -22821.177} C_VEL
LIN {X 0,Y 171.979,Z 179.147,A -85,B 0,C 180,E1 -22822.748,E2 -22822.748} C_VEL
LIN {X 0,Y 171.798,Z 178.734,A -85,B 0,C 180,E1 -22822.886,E2 -22822.886} C_VEL
LIN {X 0,Y 171.364,Z 177.134,A -85,B 0,C 180,E1 -22824.238,E2 -22824.238} C_VEL
LIN {X 0,Y 171.412,Z 177.13,A -85,B 0,C 180,E1 -22829.426,E2 -22829.426} C_VEL
LIN {X 0,Y 171.429,Z 177.129,A -85,B 0,C 180,E1 -22834.407,E2 -22834.407} C_VEL
LIN {X 0,Y 171.501,Z 177.121,A -85,B 0,C 180,E1 -22840.863,E2 -22840.863} C_VEL
LIN {X 0,Y 171.531,Z 177.116,A -85,B 0,C 180,E1 -22845.769,E2 -22845.769} C_VEL
LIN {X 0,Y 171.834,Z 177.06,A -85,B 0,C 180,E1 -22850.584,E2 -22850.584} C_VEL
LIN {X 0,Y 171.768,Z 177.079,A -85,B 0,C 180,E1 -22855.306,E2 -22855.306} C_VEL
LIN {X 0,Y 172.301,Z 177.017,A -85,B 0,C 180,E1 -22860,E2 -22860} C_VEL
LIN {X 0,Y 171.774,Z 177.064,A -85,B 0,C 180,E1 -22864.694,E2 -22864.694} C_VEL
LIN {X 0,Y 171.837,Z 177.079,A -85,B 0,C 180,E1 -22869.416,E2 -22869.416} C_VEL
LIN {X 0,Y 171.53,Z 177.105,A -85,B 0,C 180,E1 -22874.231,E2 -22874.231} C_VEL
LIN {X 0,Y 171.473,Z 177.105,A -85,B 0,C 180,E1 -22879.5,E2 -22879.5} C_VEL
LIN {X 0,Y 171.437,Z 177.112,A -85,B 0,C 180,E1 -22885.598,E2 -22885.598} C_VEL
LIN {X 0,Y 171.412,Z 177.122,A -85,B 0,C 180,E1 -22890.574,E2 -22890.574} C_VEL
LIN {X 0,Y 171.368,Z 177.139,A -85,B 0,C 180,E1 -22896.489,E2 -22896.489} C_VEL
LIN {X 0,Y 171.367,Z 177.149,A -85,B 0,C 180,E1 -22897.408,E2 -22897.408} C_VEL
LIN {X 0,Y 172.252,Z 179.789,A -85,B 0,C 180,E1 -22897.972,E2 -22897.972} C_VEL
LIN {X 0,Y 174.119,Z 181.941,A -85,B 0,C 180,E1 -22898.899,E2 -22898.899} C_VEL
LIN {X 0,Y 175.024,Z 182.675,A -85,B 0,C 180,E1 -22899.315,E2 -22899.315} C_VEL
LIN {X 0,Y 177.103,Z 186.03,A -85,B 0,C 180,E1 -22900.345,E2 -22900.345} C_VEL
LIN {X 0,Y 178.591,Z 187.767,A -85,B 0,C 180,E1 -22901.015,E2 -22901.015} C_VEL
LIN {X 0,Y 181.345,Z 191.537,A -85,B 0,C 180,E1 -22902.234,E2 -22902.234} C_VEL
LIN {X 0,Y 189.194,Z 203.358,A -85,B 0,C 180,E1 -22905.438,E2 -22905.438} C_VEL
LIN {X 0,Y 196.215,Z 215.425,A -85,B 0,C 180,E1 -22908.029,E2 -22908.029} C_VEL
LIN {X 0,Y 200.125,Z 223.384,A -85,B 0,C 180,E1 -22909.409,E2 -22909.409} C_VEL
LIN {X 0,Y 202.256,Z 228.564,A -85,B 0,C 180,E1 -22910.166,E2 -22910.166} C_VEL
LIN {X 0,Y 199.584,Z 277.629,A -85,B 0,C 180,E1 -22911.83,E2 -22911.83} C_VEL
LIN {X 0,Y 198.105,Z 290.535,A -85,B 0,C 180,E1 -22912.598,E2 -22912.598} C_VEL
LIN {X 0,Y 196.004,Z 303.178,A -85,B 0,C 180,E1 -22913.729,E2 -22913.729} C_VEL
LIN {X 0,Y 193.66,Z 314.458,A -85,B 0,C 180,E1 -22915.142,E2 -22915.142} C_VEL
LIN {X 0,Y 190.441,Z 326.078,A -85,B 0,C 180,E1 -22917.023,E2 -22917.023} C_VEL
LIN {X 0,Y 187.159,Z 336.509,A -85,B 0,C 180,E1 -22919.229,E2 -22919.229} C_VEL
LIN {X 0,Y 184.423,Z 344.7,A -85,B 0,C 180,E1 -22921.441,E2 -22921.441} C_VEL
LIN {X 0,Y 181.233,Z 352.874,A -85,B 0,C 180,E1 -22924.136,E2 -22924.136} C_VEL
LIN {X 0,Y 177.891,Z 360.544,A -85,B 0,C 180,E1 -22927.346,E2 -22927.346} C_VEL
LIN {X 0,Y 174.803,Z 367.58,A -85,B 0,C 180,E1 -22931.239,E2 -22931.239} C_VEL
LIN {X 0,Y 172.664,Z 372.264,A -85,B 0,C 180,E1 -22934.66,E2 -22934.66} C_VEL
LIN {X 0,Y 171.053,Z 375.844,A -85,B 0,C 180,E1 -22938.147,E2 -22938.147} C_VEL
LIN {X 0,Y 170.291,Z 377.69,A -85,B 0,C 180,E1 -22940.499,E2 -22940.499} C_VEL
LIN {X 0,Y 169.505,Z 379.749,A -85,B 0,C 180,E1 -22944.321,E2 -22944.321} C_VEL
LIN {X 0,Y 169.196,Z 380.665,A -85,B 0,C 180,E1 -22947.621,E2 -22947.621} C_VEL
LIN {X 0,Y 169.151,Z 380.891,A -85,B 0,C 180,E1 -22950.001,E2 -22950.001} C_VEL
LIN {X 0,Y 169.195,Z 380.697,A -85,B 0,C 180,E1 -22952.382,E2 -22952.382} C_VEL
LIN {X 0,Y 169.782,Z 379.147,A -85,B 0,C 180,E1 -22957.135,E2 -22957.135} C_VEL
LIN {X 0,Y 170.289,Z 377.795,A -85,B 0,C 180,E1 -22959.503,E2 -22959.503} C_VEL
LIN {X 0,Y 171.487,Z 374.934,A -85,B 0,C 180,E1 -22963.028,E2 -22963.028} C_VEL
LIN {X 0,Y 173.272,Z 371.047,A -85,B 0,C 180,E1 -22966.495,E2 -22966.495} C_VEL
LIN {X 0,Y 175.544,Z 366.032,A -85,B 0,C 180,E1 -22969.896,E2 -22969.896} C_VEL
LIN {X 0,Y 178.371,Z 359.711,A -85,B 0,C 180,E1 -22973.205,E2 -22973.205} C_VEL
LIN {X 0,Y 181.763,Z 351.798,A -85,B 0,C 180,E1 -22976.402,E2 -22976.402} C_VEL
LIN {X 0,Y 184.765,Z 343.851,A -85,B 0,C 180,E1 -22978.971,E2 -22978.971} C_VEL
LIN {X 0,Y 188.143,Z 333.892,A -85,B 0,C 180,E1 -22981.532,E2 -22981.532} C_VEL
LIN {X 0,Y 191.558,Z 322.796,A -85,B 0,C 180,E1 -22983.706,E2 -22983.706} C_VEL
LIN {X 0,Y 194.363,Z 311.916,A -85,B 0,C 180,E1 -22985.349,E2 -22985.349} C_VEL
LIN {X 0,Y 196.818,Z 299.887,A -85,B 0,C 180,E1 -22986.735,E2 -22986.735} C_VEL
LIN {X 0,Y 198.763,Z 286.859,A -85,B 0,C 180,E1 -22987.801,E2 -22987.801} C_VEL
LIN {X 0,Y 200.039,Z 273.921,A -85,B 0,C 180,E1 -22988.454,E2 -22988.454} C_VEL
LIN {X 0,Y 202.385,Z 228.72,A -85,B 0,C 180,E1 -22989.972,E2 -22989.972} C_VEL
LIN {X 0,Y 198.153,Z 219.03,A -85,B 0,C 180,E1 -22991.474,E2 -22991.474} C_VEL
LIN {X 0,Y 192.367,Z 208.576,A -85,B 0,C 180,E1 -22993.556,E2 -22993.556} C_VEL
LIN {X 0,Y 186.296,Z 198.881,A -85,B 0,C 180,E1 -22995.9,E2 -22995.9} C_VEL
LIN {X 0,Y 180.813,Z 190.946,A -85,B 0,C 180,E1 -22998.202,E2 -22998.202} C_VEL
LIN {X 0,Y 177.912,Z 186.838,A -85,B 0,C 180,E1 -22999.517,E2 -22999.517} C_VEL
LIN {X 0,Y 175.491,Z 183.636,A -85,B 0,C 180,E1 -23000.664,E2 -23000.664} C_VEL
LIN {X 0,Y 174.756,Z 182.335,A -85,B 0,C 180,E1 -23001.044,E2 -23001.044} C_VEL
LIN {X 0,Y 172.549,Z 180.275,A -85,B 0,C 180,E1 -23002.105,E2 -23002.105} C_VEL
LIN {X 0,Y 171.508,Z 177.883,A -85,B 0,C 180,E1 -23002.72,E2 -23002.72} C_VEL
LIN {X 0,Y 171.366,Z 177.134,A -85,B 0,C 180,E1 -23002.961,E2 -23002.961} C_VEL
LIN {X 0,Y 171.41,Z 177.133,A -85,B 0,C 180,E1 -23007.79,E2 -23007.79} C_VEL
LIN {X 0,Y 171.41,Z 177.114,A -85,B 0,C 180,E1 -23010.527,E2 -23010.527} C_VEL
LIN {X 0,Y 171.439,Z 177.116,A -85,B 0,C 180,E1 -23015.799,E2 -23015.799} C_VEL
LIN {X 0,Y 171.51,Z 177.122,A -85,B 0,C 180,E1 -23020.863,E2 -23020.863} C_VEL
LIN {X 0,Y 171.544,Z 177.092,A -85,B 0,C 180,E1 -23025.77,E2 -23025.77} C_VEL
LIN {X 0,Y 171.844,Z 177.069,A -85,B 0,C 180,E1 -23030.584,E2 -23030.584} C_VEL
LIN {X 0,Y 171.781,Z 177.075,A -85,B 0,C 180,E1 -23035.306,E2 -23035.306} C_VEL
LIN {X 0,Y 172.309,Z 176.997,A -85,B 0,C 180,E1 -23040,E2 -23040} C_VEL
LIN {X 0,Y 171.853,Z 177.067,A -85,B 0,C 180,E1 -23047.047,E2 -23047.047} C_VEL
LIN {X 0,Y 171.759,Z 177.07,A -85,B 0,C 180,E1 -23050.878,E2 -23050.878} C_VEL
LIN {X 0,Y 171.495,Z 177.098,A -85,B 0,C 180,E1 -23056.67,E2 -23056.67} C_VEL
LIN {X 0,Y 171.479,Z 177.122,A -85,B 0,C 180,E1 -23059.498,E2 -23059.498} C_VEL
LIN {X 0,Y 171.404,Z 177.131,A -85,B 0,C 180,E1 -23065.569,E2 -23065.569} C_VEL
LIN {X 0,Y 171.418,Z 177.125,A -85,B 0,C 180,E1 -23070.572,E2 -23070.572} C_VEL
LIN {X 0,Y 171.417,Z 177.28,A -85,B 0,C 180,E1 -23075.749,E2 -23075.749} C_VEL
LIN {X 0,Y 171.937,Z 179.049,A -85,B 0,C 180,E1 -23077.079,E2 -23077.079} C_VEL
LIN {X 0,Y 175.179,Z 183.952,A -85,B 0,C 180,E1 -23078.763,E2 -23078.763} C_VEL
LIN {X 0,Y 180.098,Z 191.691,A -85,B 0,C 180,E1 -23081.117,E2 -23081.117} C_VEL
LIN {X 0,Y 183.767,Z 197.944,A -85,B 0,C 180,E1 -23082.752,E2 -23082.752} C_VEL
LIN {X 0,Y 189.907,Z 209.125,A -85,B 0,C 180,E1 -23085.288,E2 -23085.288} C_VEL
LIN {X 0,Y 195.731,Z 221.68,A -85,B 0,C 180,E1 -23087.551,E2 -23087.551} C_VEL
LIN {X 0,Y 200.475,Z 233.686,A -85,B 0,C 180,E1 -23089.325,E2 -23089.325} C_VEL
LIN {X 0,Y 201.604,Z 244.261,A -85,B 0,C 180,E1 -23090.079,E2 -23090.079} C_VEL
LIN {X 0,Y 199.119,Z 289.14,A -85,B 0,C 180,E1 -23091.601,E2 -23091.601} C_VEL
LIN {X 0,Y 197.533,Z 302.263,A -85,B 0,C 180,E1 -23092.369,E2 -23092.369} C_VEL
LIN {X 0,Y 195.285,Z 314.441,A -85,B 0,C 180,E1 -23093.411,E2 -23093.411} C_VEL
LIN {X 0,Y 192.331,Z 326.626,A -85,B 0,C 180,E1 -23094.863,E2 -23094.863} C_VEL
LIN {X 0,Y 191.747,Z 328.837,A -85,B 0,C 180,E1 -23095.187,E2 -23095.187} C_VEL
LIN {X 0,Y 189.768,Z 333.934,A -85,B 0,C 180,E1 -23095.871,E2 -23095.871} C_VEL
LIN {X 0,Y 184.805,Z 341.921,A -85,B 0,C 180,E1 -23096.86,E2 -23096.86} C_VEL
LIN {X 0,Y 179.646,Z 349.416,A -85,B 0,C 180,E1 -23098.097,E2 -23098.097} C_VEL
LIN {X 0,Y 177.403,Z 353.735,A -85,B 0,C 180,E1 -23099.168,E2 -23099.168} C_VEL
LIN {X 0,Y 173.522,Z 363.244,A -85,B 0,C 180,E1 -23102.239,E2 -23102.239} C_VEL
LIN {X 0,Y 170.157,Z 371.267,A -85,B 0,C 180,E1 -23105.604,E2 -23105.604} C_VEL
LIN {X 0,Y 167.262,Z 377.698,A -85,B 0,C 180,E1 -23109.074,E2 -23109.074} C_VEL
LIN {X 0,Y 164.963,Z 382.811,A -85,B 0,C 180,E1 -23112.648,E2 -23112.648} C_VEL
LIN {X 0,Y 163.348,Z 386.79,A -85,B 0,C 180,E1 -23116.311,E2 -23116.311} C_VEL
LIN {X 0,Y 162.352,Z 389.738,A -85,B 0,C 180,E1 -23120.028,E2 -23120.028} C_VEL
LIN {X 0,Y 161.794,Z 392.147,A -85,B 0,C 180,E1 -23125.015,E2 -23125.015} C_VEL
LIN {X 0,Y 161.866,Z 392.766,A -85,B 0,C 180,E1 -23127.51,E2 -23127.51} C_VEL
LIN {X 0,Y 161.982,Z 392.983,A -85,B 0,C 180,E1 -23129.999,E2 -23129.999} C_VEL
LIN {X 0,Y 161.829,Z 392.7,A -85,B 0,C 180,E1 -23132.74,E2 -23132.74} C_VEL
LIN {X 0,Y 161.967,Z 391.11,A -85,B 0,C 180,E1 -23137.478,E2 -23137.478} C_VEL
LIN {X 0,Y 162.359,Z 389.692,A -85,B 0,C 180,E1 -23139.969,E2 -23139.969} C_VEL
LIN {X 0,Y 163.347,Z 386.724,A -85,B 0,C 180,E1 -23143.687,E2 -23143.687} C_VEL
LIN {X 0,Y 164.961,Z 382.72,A -85,B 0,C 180,E1 -23147.35,E2 -23147.35} C_VEL
LIN {X 0,Y 167.685,Z 376.575,A -85,B 0,C 180,E1 -23151.512,E2 -23151.512} C_VEL
LIN {X 0,Y 170.186,Z 371.114,A -85,B 0,C 180,E1 -23154.389,E2 -23154.389} C_VEL
LIN {X 0,Y 173.516,Z 363.055,A -85,B 0,C 180,E1 -23157.76,E2 -23157.76} C_VEL
LIN {X 0,Y 176.865,Z 354.852,A -85,B 0,C 180,E1 -23160.438,E2 -23160.438} C_VEL
LIN {X 0,Y 180.648,Z 344.854,A -85,B 0,C 180,E1 -23163,E2 -23163} C_VEL
LIN {X 0,Y 184.351,Z 333.552,A -85,B 0,C 180,E1 -23165.21,E2 -23165.21} C_VEL
LIN {X 0,Y 187.507,Z 322.483,A -85,B 0,C 180,E1 -23166.846,E2 -23166.846} C_VEL
LIN {X 0,Y 190.332,Z 310.199,A -85,B 0,C 180,E1 -23168.204,E2 -23168.204} C_VEL
LIN {X 0,Y 192.593,Z 296.599,A -85,B 0,C 180,E1 -23169.234,E2 -23169.234} C_VEL
LIN {X 0,Y 193.819,Z 283.646,A -85,B 0,C 180,E1 -23169.872,E2 -23169.872} C_VEL
LIN {X 0,Y 196.008,Z 245.277,A -85,B 0,C 180,E1 -23171.152,E2 -23171.152} C_VEL
LIN {X 0,Y 195.02,Z 235.99,A -85,B 0,C 180,E1 -23171.85,E2 -23171.85} C_VEL
LIN {X 0,Y 189.625,Z 222.366,A -85,B 0,C 180,E1 -23174.008,E2 -23174.008} C_VEL
LIN {X 0,Y 184.641,Z 211.805,A -85,B 0,C 180,E1 -23176.08,E2 -23176.08} C_VEL
LIN {X 0,Y 179.451,Z 202.182,A -85,B 0,C 180,E1 -23178.373,E2 -23178.373} C_VEL
LIN {X 0,Y 174.586,Z 193.939,A -85,B 0,C 180,E1 -23180.703,E2 -23180.703} C_VEL
LIN {X 0,Y 171.545,Z 189.124,A -85,B 0,C 180,E1 -23182.268,E2 -23182.268} C_VEL
LIN {X 0,Y 168.088,Z 183.902,A -85,B 0,C 180,E1 -23184.171,E2 -23184.171} C_VEL
LIN {X 0,Y 165.087,Z 180.449,A -85,B 0,C 180,E1 -23185.884,E2 -23185.884} C_VEL
LIN {X 0,Y 164.356,Z 178.232,A -85,B 0,C 180,E1 -23186.493,E2 -23186.493} C_VEL
LIN {X 0,Y 164.355,Z 177.999,A -85,B 0,C 180,E1 -23187.63,E2 -23187.63} C_VEL
LIN {X 0,Y 164.358,Z 178.008,A -85,B 0,C 180,E1 -23193.888,E2 -23193.888} C_VEL
LIN {X 0,Y 164.41,Z 178.005,A -85,B 0,C 180,E1 -23200.117,E2 -23200.117} C_VEL
LIN {X 0,Y 164.46,Z 177.987,A -85,B 0,C 180,E1 -23205.143,E2 -23205.143} C_VEL
LIN {X 0,Y 164.755,Z 177.94,A -85,B 0,C 180,E1 -23210.176,E2 -23210.176} C_VEL
LIN {X 0,Y 164.808,Z 177.95,A -85,B 0,C 180,E1 -23212.65,E2 -23212.65} C_VEL
LIN {X 0,Y 165.266,Z 177.893,A -85,B 0,C 180,E1 -23220,E2 -23220} C_VEL
LIN {X 0,Y 164.813,Z 177.947,A -85,B 0,C 180,E1 -23227.35,E2 -23227.35} C_VEL
LIN {X 0,Y 164.691,Z 177.953,A -85,B 0,C 180,E1 -23231.05,E2 -23231.05} C_VEL
LIN {X 0,Y 164.422,Z 177.997,A -85,B 0,C 180,E1 -23237.41,E2 -23237.41} C_VEL
LIN {X 0,Y 164.414,Z 177.984,A -85,B 0,C 180,E1 -23239.997,E2 -23239.997} C_VEL
LIN {X 0,Y 164.364,Z 177.992,A -85,B 0,C 180,E1 -23246.117,E2 -23246.117} C_VEL
LIN {X 0,Y 164.348,Z 177.999,A -85,B 0,C 180,E1 -23251.216,E2 -23251.216} C_VEL
LIN {X 0,Y 164.311,Z 178.044,A -85,B 0,C 180,E1 -23254.093,E2 -23254.093} C_VEL
LIN {X 0,Y 165.161,Z 180.537,A -85,B 0,C 180,E1 -23254.719,E2 -23254.719} C_VEL
LIN {X 0,Y 167.103,Z 182.815,A -85,B 0,C 180,E1 -23255.843,E2 -23255.843} C_VEL
LIN {X 0,Y 168.232,Z 183.712,A -85,B 0,C 180,E1 -23256.441,E2 -23256.441} C_VEL
LIN {X 0,Y 170.271,Z 187.035,A -85,B 0,C 180,E1 -23257.597,E2 -23257.597} C_VEL
LIN {X 0,Y 172.14,Z 189.133,A -85,B 0,C 180,E1 -23258.544,E2 -23258.544} C_VEL
LIN {X 0,Y 174.787,Z 192.704,A -85,B 0,C 180,E1 -23259.857,E2 -23259.857} C_VEL
LIN {X 0,Y 181.006,Z 201.792,A -85,B 0,C 180,E1 -23262.709,E2 -23262.709} C_VEL
LIN {X 0,Y 187.395,Z 212.018,A -85,B 0,C 180,E1 -23265.349,E2 -23265.349} C_VEL
LIN {X 0,Y 193.171,Z 222.534,A -85,B 0,C 180,E1 -23267.557,E2 -23267.557} C_VEL
LIN {X 0,Y 196.812,Z 230.793,A -85,B 0,C 180,E1 -23268.923,E2 -23268.923} C_VEL
LIN {X 0,Y 194.03,Z 278.287,A -85,B 0,C 180,E1 -23270.558,E2 -23270.558} C_VEL
LIN {X 0,Y 192.419,Z 291.435,A -85,B 0,C 180,E1 -23271.361,E2 -23271.361} C_VEL
LIN {X 0,Y 190.331,Z 303.445,A -85,B 0,C 180,E1 -23272.466,E2 -23272.466} C_VEL
LIN {X 0,Y 187.897,Z 314.722,A -85,B 0,C 180,E1 -23273.908,E2 -23273.908} C_VEL
LIN {X 0,Y 184.536,Z 326.341,A -85,B 0,C 180,E1 -23275.825,E2 -23275.825} C_VEL
LIN {X 0,Y 181.092,Z 336.772,A -85,B 0,C 180,E1 -23278.079,E2 -23278.079} C_VEL
LIN {X 0,Y 178.042,Z 345.453,A -85,B 0,C 180,E1 -23280.497,E2 -23280.497} C_VEL
LIN {X 0,Y 174.891,Z 353.134,A -85,B 0,C 180,E1 -23283.125,E2 -23283.125} C_VEL
LIN {X 0,Y 171.373,Z 360.805,A -85,B 0,C 180,E1 -23286.433,E2 -23286.433} C_VEL
LIN {X 0,Y 168.929,Z 366.039,A -85,B 0,C 180,E1 -23289.292,E2 -23289.292} C_VEL
LIN {X 0,Y 166.525,Z 371.111,A -85,B 0,C 180,E1 -23292.818,E2 -23292.818} C_VEL
LIN {X 0,Y 164.631,Z 375.047,A -85,B 0,C 180,E1 -23296.422,E2 -23296.422} C_VEL
LIN {X 0,Y 163.304,Z 377.95,A -85,B 0,C 180,E1 -23300.089,E2 -23300.089} C_VEL
LIN {X 0,Y 162.399,Z 380.143,A -85,B 0,C 180,E1 -23304.476,E2 -23304.476} C_VEL
LIN {X 0,Y 162.112,Z 380.924,A -85,B 0,C 180,E1 -23307.517,E2 -23307.517} C_VEL
LIN {X 0,Y 162.061,Z 381.15,A -85,B 0,C 180,E1 -23310.001,E2 -23310.001} C_VEL
LIN {X 0,Y 162.111,Z 380.956,A -85,B 0,C 180,E1 -23312.486,E2 -23312.486} C_VEL
LIN {X 0,Y 162.755,Z 379.406,A -85,B 0,C 180,E1 -23317.444,E2 -23317.444} C_VEL
LIN {X 0,Y 163.299,Z 378.054,A -85,B 0,C 180,E1 -23319.914,E2 -23319.914} C_VEL
LIN {X 0,Y 164.563,Z 375.193,A -85,B 0,C 180,E1 -23323.586,E2 -23323.586} C_VEL
LIN {X 0,Y 166.474,Z 371.305,A -85,B 0,C 180,E1 -23327.19,E2 -23327.19} C_VEL
LIN {X 0,Y 168.88,Z 366.29,A -85,B 0,C 180,E1 -23330.717,E2 -23330.717} C_VEL
LIN {X 0,Y 171.864,Z 359.968,A -85,B 0,C 180,E1 -23334.138,E2 -23334.138} C_VEL
LIN {X 0,Y 175.433,Z 352.055,A -85,B 0,C 180,E1 -23337.433,E2 -23337.433} C_VEL
LIN {X 0,Y 178.825,Z 343.435,A -85,B 0,C 180,E1 -23340.277,E2 -23340.277} C_VEL
LIN {X 0,Y 182.151,Z 334.147,A -85,B 0,C 180,E1 -23342.696,E2 -23342.696} C_VEL
LIN {X 0,Y 185.712,Z 323.05,A -85,B 0,C 180,E1 -23344.917,E2 -23344.917} C_VEL
LIN {X 0,Y 188.622,Z 312.169,A -85,B 0,C 180,E1 -23346.596,E2 -23346.596} C_VEL
LIN {X 0,Y 191.194,Z 300.138,A -85,B 0,C 180,E1 -23348.004,E2 -23348.004} C_VEL
LIN {X 0,Y 193.158,Z 287.606,A -85,B 0,C 180,E1 -23349.056,E2 -23349.056} C_VEL
LIN {X 0,Y 194.47,Z 274.888,A -85,B 0,C 180,E1 -23349.729,E2 -23349.729} C_VEL
LIN {X 0,Y 196.899,Z 230.83,A -85,B 0,C 180,E1 -23351.235,E2 -23351.235} C_VEL
LIN {X 0,Y 193.043,Z 222.15,A -85,B 0,C 180,E1 -23352.685,E2 -23352.685} C_VEL
LIN {X 0,Y 186.798,Z 210.893,A -85,B 0,C 180,E1 -23355.093,E2 -23355.093} C_VEL
LIN {X 0,Y 180.059,Z 200.3,A -85,B 0,C 180,E1 -23357.922,E2 -23357.922} C_VEL
LIN {X 0,Y 174.349,Z 192.216,A -85,B 0,C 180,E1 -23360.576,E2 -23360.576} C_VEL
LIN {X 0,Y 171.322,Z 188.016,A -85,B 0,C 180,E1 -23362.117,E2 -23362.117} C_VEL
LIN {X 0,Y 168.956,Z 185.155,A -85,B 0,C 180,E1 -23363.369,E2 -23363.369} C_VEL
LIN {X 0,Y 167.969,Z 183.356,A -85,B 0,C 180,E1 -23363.957,E2 -23363.957} C_VEL
LIN {X 0,Y 165.582,Z 181.206,A -85,B 0,C 180,E1 -23365.279,E2 -23365.279} C_VEL
LIN {X 0,Y 164.459,Z 178.699,A -85,B 0,C 180,E1 -23366.046,E2 -23366.046} C_VEL
LIN {X 0,Y 164.325,Z 178.002,A -85,B 0,C 180,E1 -23366.22,E2 -23366.22} C_VEL
LIN {X 0,Y 164.372,Z 177.999,A -85,B 0,C 180,E1 -23369.13,E2 -23369.13} C_VEL
LIN {X 0,Y 164.396,Z 178.005,A -85,B 0,C 180,E1 -23374.69,E2 -23374.69} C_VEL
LIN {X 0,Y 164.419,Z 178,A -85,B 0,C 180,E1 -23380.117,E2 -23380.117} C_VEL
LIN {X 0,Y 164.473,Z 177.97,A -85,B 0,C 180,E1 -23385.144,E2 -23385.144} C_VEL
LIN {X 0,Y 164.765,Z 177.955,A -85,B 0,C 180,E1 -23390.176,E2 -23390.176} C_VEL
LIN {X 0,Y 164.819,Z 177.925,A -85,B 0,C 180,E1 -23392.65,E2 -23392.65} C_VEL
LIN {X 0,Y 165.273,Z 177.872,A -85,B 0,C 180,E1 -23400,E2 -23400} C_VEL
LIN {X 0,Y 164.815,Z 177.938,A -85,B 0,C 180,E1 -23407.35,E2 -23407.35} C_VEL
LIN {X 0,Y 164.697,Z 177.95,A -85,B 0,C 180,E1 -23411.047,E2 -23411.047} C_VEL
LIN {X 0,Y 164.421,Z 177.98,A -85,B 0,C 180,E1 -23417.41,E2 -23417.41} C_VEL
LIN {X 0,Y 164.42,Z 178.004,A -85,B 0,C 180,E1 -23419.996,E2 -23419.996} C_VEL
LIN {X 0,Y 164.34,Z 178.015,A -85,B 0,C 180,E1 -23426.094,E2 -23426.094} C_VEL
LIN {X 0,Y 164.373,Z 178.003,A -85,B 0,C 180,E1 -23432.368,E2 -23432.368} C_VEL
LIN {X 0,Y 164.364,Z 178.21,A -85,B 0,C 180,E1 -23433.33,E2 -23433.33} C_VEL
LIN {X 0,Y 165.526,Z 181.163,A -85,B 0,C 180,E1 -23434.22,E2 -23434.22} C_VEL
LIN {X 0,Y 168.643,Z 184.458,A -85,B 0,C 180,E1 -23435.968,E2 -23435.968} C_VEL
LIN {X 0,Y 172.105,Z 189.752,A -85,B 0,C 180,E1 -23437.867,E2 -23437.867} C_VEL
LIN {X 0,Y 176.666,Z 197.25,A -85,B 0,C 180,E1 -23440.178,E2 -23440.178} C_VEL
LIN {X 0,Y 181.118,Z 204.984,A -85,B 0,C 180,E1 -23442.252,E2 -23442.252} C_VEL
LIN {X 0,Y 187.23,Z 216.893,A -85,B 0,C 180,E1 -23444.891,E2 -23444.891} C_VEL
LIN {X 0,Y 193.103,Z 230.652,A -85,B 0,C 180,E1 -23447.284,E2 -23447.284} C_VEL
LIN {X 0,Y 195.341,Z 237.024,A -85,B 0,C 180,E1 -23448.19,E2 -23448.19} C_VEL
LIN {X 0,Y 196.132,Z 245.673,A -85,B 0,C 180,E1 -23448.807,E2 -23448.807} C_VEL
LIN {X 0,Y 193.57,Z 289.297,A -85,B 0,C 180,E1 -23450.317,E2 -23450.317} C_VEL
LIN {X 0,Y 191.831,Z 302.758,A -85,B 0,C 180,E1 -23451.126,E2 -23451.126} C_VEL
LIN {X 0,Y 189.381,Z 315.293,A -85,B 0,C 180,E1 -23452.242,E2 -23452.242} C_VEL
LIN {X 0,Y 186.116,Z 327.956,A -85,B 0,C 180,E1 -23453.841,E2 -23453.841} C_VEL
LIN {X 0,Y 182.686,Z 339.227,A -85,B 0,C 180,E1 -23455.761,E2 -23455.761} C_VEL
LIN {X 0,Y 179.085,Z 349.382,A -85,B 0,C 180,E1 -23458.008,E2 -23458.008} C_VEL
LIN {X 0,Y 177.403,Z 353.735,A -85,B 0,C 180,E1 -23459.168,E2 -23459.168} C_VEL
LIN {X 0,Y 175.169,Z 357.957,A -85,B 0,C 180,E1 -23460.336,E2 -23460.336} C_VEL
LIN {X 0,Y 167.723,Z 366.732,A -85,B 0,C 180,E1 -23462.935,E2 -23462.935} C_VEL
LIN {X 0,Y 163.901,Z 371.254,A -85,B 0,C 180,E1 -23464.737,E2 -23464.737} C_VEL
LIN {X 0,Y 162.633,Z 373.356,A -85,B 0,C 180,E1 -23465.8,E2 -23465.8} C_VEL
LIN {X 0,Y 159.785,Z 379.266,A -85,B 0,C 180,E1 -23469.397,E2 -23469.397} C_VEL
LIN {X 0,Y 157.483,Z 383.989,A -85,B 0,C 180,E1 -23473.136,E2 -23473.136} C_VEL
LIN {X 0,Y 155.997,Z 387.609,A -85,B 0,C 180,E1 -23476.981,E2 -23476.981} C_VEL
LIN {X 0,Y 155.324,Z 389.477,A -85,B 0,C 180,E1 -23479.571,E2 -23479.571} C_VEL
LIN {X 0,Y 154.905,Z 390.882,A -85,B 0,C 180,E1 -23482.176,E2 -23482.176} C_VEL
LIN {X 0,Y 154.776,Z 392.507,A -85,B 0,C 180,E1 -23487.396,E2 -23487.396} C_VEL
LIN {X 0,Y 154.891,Z 392.724,A -85,B 0,C 180,E1 -23489.999,E2 -23489.999} C_VEL
LIN {X 0,Y 154.739,Z 392.491,A -85,B 0,C 180,E1 -23492.602,E2 -23492.602} C_VEL
LIN {X 0,Y 154.746,Z 391.866,A -85,B 0,C 180,E1 -23495.21,E2 -23495.21} C_VEL
LIN {X 0,Y 154.921,Z 390.85,A -85,B 0,C 180,E1 -23497.82,E2 -23497.82} C_VEL
LIN {X 0,Y 155.331,Z 389.43,A -85,B 0,C 180,E1 -23500.425,E2 -23500.425} C_VEL
LIN {X 0,Y 156.423,Z 386.463,A -85,B 0,C 180,E1 -23504.305,E2 -23504.305} C_VEL
LIN {X 0,Y 158.185,Z 382.459,A -85,B 0,C 180,E1 -23508.118,E2 -23508.118} C_VEL
LIN {X 0,Y 161.083,Z 376.313,A -85,B 0,C 180,E1 -23512.441,E2 -23512.441} C_VEL
LIN {X 0,Y 164.073,Z 369.859,A -85,B 0,C 180,E1 -23515.904,E2 -23515.904} C_VEL
LIN {X 0,Y 167.888,Z 361.298,A -85,B 0,C 180,E1 -23519.462,E2 -23519.462} C_VEL
LIN {X 0,Y 171.503,Z 352.781,A -85,B 0,C 180,E1 -23522.188,E2 -23522.188} C_VEL
LIN {X 0,Y 175.567,Z 342.265,A -85,B 0,C 180,E1 -23524.778,E2 -23524.778} C_VEL
LIN {X 0,Y 179.043,Z 331.86,A -85,B 0,C 180,E1 -23526.768,E2 -23526.768} C_VEL
LIN {X 0,Y 182.349,Z 320.447,A -85,B 0,C 180,E1 -23528.422,E2 -23528.422} C_VEL
LIN {X 0,Y 185.072,Z 308.682,A -85,B 0,C 180,E1 -23529.674,E2 -23529.674} C_VEL
LIN {X 0,Y 187.29,Z 295.223,A -85,B 0,C 180,E1 -23530.678,E2 -23530.678} C_VEL
LIN {X 0,Y 188.468,Z 282.798,A -85,B 0,C 180,E1 -23531.279,E2 -23531.279} C_VEL
LIN {X 0,Y 190.621,Z 245.841,A -85,B 0,C 180,E1 -23532.54,E2 -23532.54} C_VEL
LIN {X 0,Y 189.845,Z 238.657,A -85,B 0,C 180,E1 -23533.115,E2 -23533.115} C_VEL
LIN {X 0,Y 184.894,Z 225.975,A -85,B 0,C 180,E1 -23535.233,E2 -23535.233} C_VEL
LIN {X 0,Y 180.562,Z 216.466,A -85,B 0,C 180,E1 -23537.161,E2 -23537.161} C_VEL
LIN {X 0,Y 174.337,Z 204.663,A -85,B 0,C 180,E1 -23540.127,E2 -23540.127} C_VEL
LIN {X 0,Y 168.622,Z 195.052,A -85,B 0,C 180,E1 -23543.145,E2 -23543.145} C_VEL
LIN {X 0,Y 164.757,Z 189.215,A -85,B 0,C 180,E1 -23545.392,E2 -23545.392} C_VEL
LIN {X 0,Y 162.217,Z 186.258,A -85,B 0,C 180,E1 -23546.933,E2 -23546.933} C_VEL
LIN {X 0,Y 161.104,Z 184.312,A -85,B 0,C 180,E1 -23547.697,E2 -23547.697} C_VEL
LIN {X 0,Y 158.762,Z 182.385,A -85,B 0,C 180,E1 -23549.21,E2 -23549.21} C_VEL
LIN {X 0,Y 157.544,Z 180.119,A -85,B 0,C 180,E1 -23550.154,E2 -23550.154} C_VEL
LIN {X 0,Y 157.237,Z 178.884,A -85,B 0,C 180,E1 -23550.55,E2 -23550.55} C_VEL
LIN {X 0,Y 157.304,Z 178.88,A -85,B 0,C 180,E1 -23553.463,E2 -23553.463} C_VEL
LIN {X 0,Y 157.354,Z 178.882,A -85,B 0,C 180,E1 -23559.702,E2 -23559.702} C_VEL
LIN {X 0,Y 157.395,Z 178.861,A -85,B 0,C 180,E1 -23564.46,E2 -23564.46} C_VEL
LIN {X 0,Y 157.678,Z 178.822,A -85,B 0,C 180,E1 -23569.73,E2 -23569.73} C_VEL
LIN {X 0,Y 157.747,Z 178.826,A -85,B 0,C 180,E1 -23572.319,E2 -23572.319} C_VEL
LIN {X 0,Y 158.228,Z 178.77,A -85,B 0,C 180,E1 -23580,E2 -23580} C_VEL
LIN {X 0,Y 157.751,Z 178.83,A -85,B 0,C 180,E1 -23587.681,E2 -23587.681} C_VEL
LIN {X 0,Y 157.621,Z 178.831,A -85,B 0,C 180,E1 -23591.218,E2 -23591.218} C_VEL
LIN {X 0,Y 157.397,Z 178.878,A -85,B 0,C 180,E1 -23595.54,E2 -23595.54} C_VEL
LIN {X 0,Y 157.303,Z 178.875,A -85,B 0,C 180,E1 -23600.942,E2 -23600.942} C_VEL
LIN {X 0,Y 157.305,Z 178.872,A -85,B 0,C 180,E1 -23606.682,E2 -23606.682} C_VEL
LIN {X 0,Y 157.28,Z 178.903,A -85,B 0,C 180,E1 -23610.13,E2 -23610.13} C_VEL
LIN {X 0,Y 158.026,Z 181.218,A -85,B 0,C 180,E1 -23610.801,E2 -23610.801} C_VEL
LIN {X 0,Y 159.977,Z 183.639,A -85,B 0,C 180,E1 -23612.169,E2 -23612.169} C_VEL
LIN {X 0,Y 161.527,Z 184.783,A -85,B 0,C 180,E1 -23613.134,E2 -23613.134} C_VEL
LIN {X 0,Y 163.442,Z 187.956,A -85,B 0,C 180,E1 -23614.403,E2 -23614.403} C_VEL
LIN {X 0,Y 165.368,Z 189.861,A -85,B 0,C 180,E1 -23615.517,E2 -23615.517} C_VEL
LIN {X 0,Y 167.798,Z 193.419,A -85,B 0,C 180,E1 -23616.925,E2 -23616.925} C_VEL
LIN {X 0,Y 169.154,Z 195.104,A -85,B 0,C 180,E1 -23617.654,E2 -23617.654} C_VEL
LIN {X 0,Y 175.162,Z 203.726,A -85,B 0,C 180,E1 -23620.693,E2 -23620.693} C_VEL
LIN {X 0,Y 181.501,Z 213.719,A -85,B 0,C 180,E1 -23623.558,E2 -23623.558} C_VEL
LIN {X 0,Y 187.504,Z 224.462,A -85,B 0,C 180,E1 -23626.038,E2 -23626.038} C_VEL
LIN {X 0,Y 190.805,Z 231.512,A -85,B 0,C 180,E1 -23627.351,E2 -23627.351} C_VEL
LIN {X 0,Y 191.432,Z 233.588,A -85,B 0,C 180,E1 -23627.63,E2 -23627.63} C_VEL
LIN {X 0,Y 188.609,Z 278.625,A -85,B 0,C 180,E1 -23629.195,E2 -23629.195} C_VEL
LIN {X 0,Y 186.917,Z 291.852,A -85,B 0,C 180,E1 -23630.017,E2 -23630.017} C_VEL
LIN {X 0,Y 184.535,Z 304.791,A -85,B 0,C 180,E1 -23631.245,E2 -23631.245} C_VEL
LIN {X 0,Y 181.699,Z 316.569,A -85,B 0,C 180,E1 -23632.819,E2 -23632.819} C_VEL
LIN {X 0,Y 178.33,Z 327.889,A -85,B 0,C 180,E1 -23634.806,E2 -23634.806} C_VEL
LIN {X 0,Y 174.749,Z 338.088,A -85,B 0,C 180,E1 -23637.118,E2 -23637.118} C_VEL
LIN {X 0,Y 171.114,Z 347.529,A -85,B 0,C 180,E1 -23639.919,E2 -23639.919} C_VEL
LIN {X 0,Y 167.291,Z 356.126,A -85,B 0,C 180,E1 -23643.155,E2 -23643.155} C_VEL
LIN {X 0,Y 163.825,Z 363.282,A -85,B 0,C 180,E1 -23646.622,E2 -23646.622} C_VEL
LIN {X 0,Y 161.411,Z 368.102,A -85,B 0,C 180,E1 -23649.617,E2 -23649.617} C_VEL
LIN {X 0,Y 159.001,Z 372.785,A -85,B 0,C 180,E1 -23653.305,E2 -23653.305} C_VEL
LIN {X 0,Y 157.184,Z 376.364,A -85,B 0,C 180,E1 -23657.083,E2 -23657.083} C_VEL
LIN {X 0,Y 156.309,Z 378.21,A -85,B 0,C 180,E1 -23659.641,E2 -23659.641} C_VEL
LIN {X 0,Y 155.721,Z 379.593,A -85,B 0,C 180,E1 -23662.22,E2 -23662.22} C_VEL
LIN {X 0,Y 155.03,Z 381.183,A -85,B 0,C 180,E1 -23667.403,E2 -23667.403} C_VEL
LIN {X 0,Y 154.972,Z 381.409,A -85,B 0,C 180,E1 -23670.001,E2 -23670.001} C_VEL
LIN {X 0,Y 155.03,Z 381.215,A -85,B 0,C 180,E1 -23672.6,E2 -23672.6} C_VEL
LIN {X 0,Y 155.722,Z 379.664,A -85,B 0,C 180,E1 -23677.783,E2 -23677.783} C_VEL
LIN {X 0,Y 156.303,Z 378.312,A -85,B 0,C 180,E1 -23680.363,E2 -23680.363} C_VEL
LIN {X 0,Y 157.667,Z 375.451,A -85,B 0,C 180,E1 -23684.193,E2 -23684.193} C_VEL
LIN {X 0,Y 159.691,Z 371.564,A -85,B 0,C 180,E1 -23687.944,E2 -23687.944} C_VEL
LIN {X 0,Y 162.259,Z 366.548,A -85,B 0,C 180,E1 -23691.604,E2 -23691.604} C_VEL
LIN {X 0,Y 165.408,Z 360.226,A -85,B 0,C 180,E1 -23695.145,E2 -23695.145} C_VEL
LIN {X 0,Y 169.163,Z 352.311,A -85,B 0,C 180,E1 -23698.541,E2 -23698.541} C_VEL
LIN {X 0,Y 172.598,Z 343.993,A -85,B 0,C 180,E1 -23701.376,E2 -23701.376} C_VEL
LIN {X 0,Y 176.228,Z 334.402,A -85,B 0,C 180,E1 -23703.941,E2 -23703.941} C_VEL
LIN {X 0,Y 179.956,Z 323.304,A -85,B 0,C 180,E1 -23706.207,E2 -23706.207} C_VEL
LIN {X 0,Y 182.979,Z 312.423,A -85,B 0,C 180,E1 -23707.919,E2 -23707.919} C_VEL
LIN {X 0,Y 185.67,Z 300.389,A -85,B 0,C 180,E1 -23709.348,E2 -23709.348} C_VEL
LIN {X 0,Y 187.715,Z 287.799,A -85,B 0,C 180,E1 -23710.422,E2 -23710.422} C_VEL
LIN {X 0,Y 189.091,Z 274.842,A -85,B 0,C 180,E1 -23711.114,E2 -23711.114} C_VEL
LIN {X 0,Y 191.62,Z 233.294,A -85,B 0,C 180,E1 -23712.522,E2 -23712.522} C_VEL
LIN {X 0,Y 187.907,Z 225.055,A -85,B 0,C 180,E1 -23714.007,E2 -23714.007} C_VEL
LIN {X 0,Y 182.123,Z 214.687,A -85,B 0,C 180,E1 -23716.387,E2 -23716.387} C_VEL
LIN {X 0,Y 176.297,Z 205.382,A -85,B 0,C 180,E1 -23718.995,E2 -23718.995} C_VEL
LIN {X 0,Y 171.003,Z 197.707,A -85,B 0,C 180,E1 -23721.605,E2 -23721.605} C_VEL
LIN {X 0,Y 167.997,Z 193.577,A -85,B 0,C 180,E1 -23723.219,E2 -23723.219} C_VEL
LIN {X 0,Y 165.478,Z 190.019,A -85,B 0,C 180,E1 -23724.675,E2 -23724.675} C_VEL
LIN {X 0,Y 162.215,Z 186.178,A -85,B 0,C 180,E1 -23726.654,E2 -23726.654} C_VEL
LIN {X 0,Y 161.21,Z 184.395,A -85,B 0,C 180,E1 -23727.351,E2 -23727.351} C_VEL
LIN {X 0,Y 158.767,Z 182.37,A -85,B 0,C 180,E1 -23728.941,E2 -23728.941} C_VEL
LIN {X 0,Y 157.462,Z 179.806,A -85,B 0,C 180,E1 -23729.976,E2 -23729.976} C_VEL
LIN {X 0,Y 157.262,Z 178.875,A -85,B 0,C 180,E1 -23730.279,E2 -23730.279} C_VEL
LIN {X 0,Y 157.311,Z 178.888,A -85,B 0,C 180,E1 -23733.464,E2 -23733.464} C_VEL
LIN {X 0,Y 157.362,Z 178.872,A -85,B 0,C 180,E1 -23739.701,E2 -23739.701} C_VEL
LIN {X 0,Y 157.407,Z 178.85,A -85,B 0,C 180,E1 -23744.461,E2 -23744.461} C_VEL
LIN {X 0,Y 157.688,Z 178.84,A -85,B 0,C 180,E1 -23749.73,E2 -23749.73} C_VEL
LIN {X 0,Y 157.758,Z 178.804,A -85,B 0,C 180,E1 -23752.319,E2 -23752.319} C_VEL
LIN {X 0,Y 158.235,Z 178.748,A -85,B 0,C 180,E1 -23760,E2 -23760} C_VEL
LIN {X 0,Y 157.754,Z 178.813,A -85,B 0,C 180,E1 -23767.681,E2 -23767.681} C_VEL
LIN {X 0,Y 157.627,Z 178.831,A -85,B 0,C 180,E1 -23771.215,E2 -23771.215} C_VEL
LIN {X 0,Y 157.397,Z 178.856,A -85,B 0,C 180,E1 -23775.54,E2 -23775.54} C_VEL
LIN {X 0,Y 157.304,Z 178.885,A -85,B 0,C 180,E1 -23780.942,E2 -23780.942} C_VEL
LIN {X 0,Y 157.268,Z 178.894,A -85,B 0,C 180,E1 -23786.649,E2 -23786.649} C_VEL
LIN {X 0,Y 157.258,Z 179.025,A -85,B 0,C 180,E1 -23789.354,E2 -23789.354} C_VEL
LIN {X 0,Y 158.097,Z 181.438,A -85,B 0,C 180,E1 -23790.099,E2 -23790.099} C_VEL
LIN {X 0,Y 160.236,Z 183.791,A -85,B 0,C 180,E1 -23791.578,E2 -23791.578} C_VEL
LIN {X 0,Y 161.531,Z 184.791,A -85,B 0,C 180,E1 -23792.391,E2 -23792.391} C_VEL
LIN {X 0,Y 163.384,Z 187.846,A -85,B 0,C 180,E1 -23793.63,E2 -23793.63} C_VEL
LIN {X 0,Y 165.839,Z 190.615,A -85,B 0,C 180,E1 -23795.077,E2 -23795.077} C_VEL
LIN {X 0,Y 169.783,Z 196.988,A -85,B 0,C 180,E1 -23797.35,E2 -23797.35} C_VEL
LIN {X 0,Y 173.121,Z 202.481,A -85,B 0,C 180,E1 -23799.117,E2 -23799.117} C_VEL
LIN {X 0,Y 177.698,Z 210.831,A -85,B 0,C 180,E1 -23801.383,E2 -23801.383} C_VEL
LIN {X 0,Y 182.897,Z 221.202,A -85,B 0,C 180,E1 -23803.762,E2 -23803.762} C_VEL
LIN {X 0,Y 188.344,Z 234.273,A -85,B 0,C 180,E1 -23806.131,E2 -23806.131} C_VEL
LIN {X 0,Y 190.239,Z 239.789,A -85,B 0,C 180,E1 -23806.952,E2 -23806.952} C_VEL
LIN {X 0,Y 190.764,Z 247.076,A -85,B 0,C 180,E1 -23807.462,E2 -23807.462} C_VEL
LIN {X 0,Y 188.186,Z 288.823,A -85,B 0,C 180,E1 -23808.926,E2 -23808.926} C_VEL
LIN {X 0,Y 186.419,Z 302.196,A -85,B 0,C 180,E1 -23809.736,E2 -23809.736} C_VEL
LIN {X 0,Y 183.82,Z 315.04,A -85,B 0,C 180,E1 -23810.887,E2 -23810.887} C_VEL
LIN {X 0,Y 180.432,Z 327.701,A -85,B 0,C 180,E1 -23812.51,E2 -23812.51} C_VEL
LIN {X 0,Y 176.862,Z 338.972,A -85,B 0,C 180,E1 -23814.467,E2 -23814.467} C_VEL
LIN {X 0,Y 173.087,Z 349.125,A -85,B 0,C 180,E1 -23816.759,E2 -23816.759} C_VEL
LIN {X 0,Y 169.297,Z 358.279,A -85,B 0,C 180,E1 -23819.433,E2 -23819.433} C_VEL
LIN {X 0,Y 165.414,Z 367.215,A -85,B 0,C 180,E1 -23822.823,E2 -23822.823} C_VEL
LIN {X 0,Y 162.633,Z 373.356,A -85,B 0,C 180,E1 -23825.8,E2 -23825.8} C_VEL
LIN {X 0,Y 160.583,Z 376.394,A -85,B 0,C 180,E1 -23827.446,E2 -23827.446} C_VEL
LIN {X 0,Y 155.645,Z 380.821,A -85,B 0,C 180,E1 -23830.126,E2 -23830.126} C_VEL
LIN {X 0,Y 150.992,Z 384.508,A -85,B 0,C 180,E1 -23833.101,E2 -23833.101} C_VEL
LIN {X 0,Y 149.451,Z 386.384,A -85,B 0,C 180,E1 -23835.157,E2 -23835.157} C_VEL
LIN {X 0,Y 148.318,Z 389.218,A -85,B 0,C 180,E1 -23839.073,E2 -23839.073} C_VEL
LIN {X 0,Y 147.631,Z 391.629,A -85,B 0,C 180,E1 -23844.535,E2 -23844.535} C_VEL
LIN {X 0,Y 147.679,Z 392.349,A -85,B 0,C 180,E1 -23847.992,E2 -23847.992} C_VEL
LIN {X 0,Y 147.79,Z 392.465,A -85,B 0,C 180,E1 -23849.999,E2 -23849.999} C_VEL
LIN {X 0,Y 147.644,Z 392.231,A -85,B 0,C 180,E1 -23852.727,E2 -23852.727} C_VEL
LIN {X 0,Y 147.679,Z 391.606,A -85,B 0,C 180,E1 -23855.46,E2 -23855.46} C_VEL
LIN {X 0,Y 147.871,Z 390.59,A -85,B 0,C 180,E1 -23858.196,E2 -23858.196} C_VEL
LIN {X 0,Y 148.324,Z 389.169,A -85,B 0,C 180,E1 -23860.924,E2 -23860.924} C_VEL
LIN {X 0,Y 149.5,Z 386.201,A -85,B 0,C 180,E1 -23864.983,E2 -23864.983} C_VEL
LIN {X 0,Y 151.414,Z 382.197,A -85,B 0,C 180,E1 -23868.958,E2 -23868.958} C_VEL
LIN {X 0,Y 154.534,Z 376.052,A -85,B 0,C 180,E1 -23873.447,E2 -23873.447} C_VEL
LIN {X 0,Y 157.759,Z 369.472,A -85,B 0,C 180,E1 -23877.095,E2 -23877.095} C_VEL
LIN {X 0,Y 161.716,Z 361.036,A -85,B 0,C 180,E1 -23880.705,E2 -23880.705} C_VEL
LIN {X 0,Y 165.522,Z 352.518,A -85,B 0,C 180,E1 -23883.501,E2 -23883.501} C_VEL
LIN {X 0,Y 169.78,Z 342.002,A -85,B 0,C 180,E1 -23886.146,E2 -23886.146} C_VEL
LIN {X 0,Y 173.408,Z 331.596,A -85,B 0,C 180,E1 -23888.172,E2 -23888.172} C_VEL
LIN {X 0,Y 176.844,Z 320.182,A -85,B 0,C 180,E1 -23889.851,E2 -23889.851} C_VEL
LIN {X 0,Y 179.65,Z 308.414,A -85,B 0,C 180,E1 -23891.123,E2 -23891.123} C_VEL
LIN {X 0,Y 181.996,Z 294.611,A -85,B 0,C 180,E1 -23892.161,E2 -23892.161} C_VEL
LIN {X 0,Y 183.195,Z 282.086,A -85,B 0,C 180,E1 -23892.769,E2 -23892.769} C_VEL
LIN {X 0,Y 185.392,Z 246.874,A -85,B 0,C 180,E1 -23893.972,E2 -23893.972} C_VEL
LIN {X 0,Y 184.801,Z 241.292,A -85,B 0,C 180,E1 -23894.443,E2 -23894.443} C_VEL
LIN {X 0,Y 179.98,Z 228.851,A -85,B 0,C 180,E1 -23896.653,E2 -23896.653} C_VEL
LIN {X 0,Y 175.708,Z 219.394,A -85,B 0,C 180,E1 -23898.702,E2 -23898.702} C_VEL
LIN {X 0,Y 170.069,Z 208.637,A -85,B 0,C 180,E1 -23901.598,E2 -23901.598} C_VEL
LIN {X 0,Y 165.206,Z 200.252,A -85,B 0,C 180,E1 -23904.361,E2 -23904.361} C_VEL
LIN {X 0,Y 162.025,Z 195.249,A -85,B 0,C 180,E1 -23906.331,E2 -23906.331} C_VEL
LIN {X 0,Y 159.367,Z 191.957,A -85,B 0,C 180,E1 -23908.049,E2 -23908.049} C_VEL
LIN {X 0,Y 158.431,Z 190.531,A -85,B 0,C 180,E1 -23908.711,E2 -23908.711} C_VEL
LIN {X 0,Y 155.843,Z 187.844,A -85,B 0,C 180,E1 -23910.539,E2 -23910.539} C_VEL
LIN {X 0,Y 154.495,Z 185.441,A -85,B 0,C 180,E1 -23911.653,E2 -23911.653} C_VEL
LIN {X 0,Y 152.01,Z 183.623,A -85,B 0,C 180,E1 -23913.607,E2 -23913.607} C_VEL
LIN {X 0,Y 150.575,Z 181.308,A -85,B 0,C 180,E1 -23914.967,E2 -23914.967} C_VEL
LIN {X 0,Y 150.214,Z 179.762,A -85,B 0,C 180,E1 -23915.466,E2 -23915.466} C_VEL
LIN {X 0,Y 150.291,Z 179.761,A -85,B 0,C 180,E1 -23920.893,E2 -23920.893} C_VEL
LIN {X 0,Y 150.395,Z 179.751,A -85,B 0,C 180,E1 -23926.488,E2 -23926.488} C_VEL
LIN {X 0,Y 150.598,Z 179.705,A -85,B 0,C 180,E1 -23929.242,E2 -23929.242} C_VEL
LIN {X 0,Y 150.671,Z 179.702,A -85,B 0,C 180,E1 -23931.956,E2 -23931.956} C_VEL
LIN {X 0,Y 151.188,Z 179.645,A -85,B 0,C 180,E1 -23940,E2 -23940} C_VEL
LIN {X 0,Y 150.69,Z 179.712,A -85,B 0,C 180,E1 -23948.043,E2 -23948.043} C_VEL
LIN {X 0,Y 150.565,Z 179.707,A -85,B 0,C 180,E1 -23951.423,E2 -23951.423} C_VEL
LIN {X 0,Y 150.304,Z 179.763,A -85,B 0,C 180,E1 -23956.293,E2 -23956.293} C_VEL
LIN {X 0,Y 150.278,Z 179.747,A -85,B 0,C 180,E1 -23960.724,E2 -23960.724} C_VEL
LIN {X 0,Y 150.232,Z 179.934,A -85,B 0,C 180,E1 -23965.161,E2 -23965.161} C_VEL
LIN {X 0,Y 151.037,Z 182.269,A -85,B 0,C 180,E1 -23966.063,E2 -23966.063} C_VEL
LIN {X 0,Y 153.127,Z 184.676,A -85,B 0,C 180,E1 -23967.877,E2 -23967.877} C_VEL
LIN {X 0,Y 154.78,Z 185.719,A -85,B 0,C 180,E1 -23969.124,E2 -23969.124} C_VEL
LIN {X 0,Y 156.708,Z 188.978,A -85,B 0,C 180,E1 -23970.669,E2 -23970.669} C_VEL
LIN {X 0,Y 158.972,Z 191.181,A -85,B 0,C 180,E1 -23972.218,E2 -23972.218} C_VEL
LIN {X 0,Y 161.471,Z 194.734,A -85,B 0,C 180,E1 -23973.894,E2 -23973.894} C_VEL
LIN {X 0,Y 162.773,Z 196.28,A -85,B 0,C 180,E1 -23974.696,E2 -23974.696} C_VEL
LIN {X 0,Y 165.49,Z 199.935,A -85,B 0,C 180,E1 -23976.311,E2 -23976.311} C_VEL
LIN {X 0,Y 171.821,Z 209.275,A -85,B 0,C 180,E1 -23979.726,E2 -23979.726} C_VEL
LIN {X 0,Y 177.637,Z 218.693,A -85,B 0,C 180,E1 -23982.512,E2 -23982.512} C_VEL
LIN {X 0,Y 183.284,Z 229.067,A -85,B 0,C 180,E1 -23984.99,E2 -23984.99} C_VEL
LIN {X 0,Y 186.064,Z 235.055,A -85,B 0,C 180,E1 -23986.165,E2 -23986.165} C_VEL
LIN {X 0,Y 183.3,Z 278.899,A -85,B 0,C 180,E1 -23987.746,E2 -23987.746} C_VEL
LIN {X 0,Y 181.475,Z 292.681,A -85,B 0,C 180,E1 -23988.629,E2 -23988.629} C_VEL
LIN {X 0,Y 179.071,Z 305.056,A -85,B 0,C 180,E1 -23989.828,E2 -23989.828} C_VEL
LIN {X 0,Y 176.105,Z 316.833,A -85,B 0,C 180,E1 -23991.425,E2 -23991.425} C_VEL
LIN {X 0,Y 172.578,Z 328.153,A -85,B 0,C 180,E1 -23993.448,E2 -23993.448} C_VEL
LIN {X 0,Y 168.826,Z 338.351,A -85,B 0,C 180,E1 -23995.809,E2 -23995.809} C_VEL
LIN {X 0,Y 164.919,Z 348.014,A -85,B 0,C 180,E1 -23998.763,E2 -23998.763} C_VEL
LIN {X 0,Y 161,Z 356.387,A -85,B 0,C 180,E1 -24002.016,E2 -24002.016} C_VEL
LIN {X 0,Y 157.335,Z 363.543,A -85,B 0,C 180,E1 -24005.597,E2 -24005.597} C_VEL
LIN {X 0,Y 154.779,Z 368.363,A -85,B 0,C 180,E1 -24008.702,E2 -24008.702} C_VEL
LIN {X 0,Y 152.205,Z 373.046,A -85,B 0,C 180,E1 -24012.536,E2 -24012.536} C_VEL
LIN {X 0,Y 150.287,Z 376.624,A -85,B 0,C 180,E1 -24016.48,E2 -24016.48} C_VEL
LIN {X 0,Y 149.343,Z 378.469,A -85,B 0,C 180,E1 -24019.152,E2 -24019.152} C_VEL
LIN {X 0,Y 148.686,Z 379.853,A -85,B 0,C 180,E1 -24021.849,E2 -24021.849} C_VEL
LIN {X 0,Y 147.94,Z 381.443,A -85,B 0,C 180,E1 -24027.279,E2 -24027.279} C_VEL
LIN {X 0,Y 147.886,Z 381.668,A -85,B 0,C 180,E1 -24030.001,E2 -24030.001} C_VEL
LIN {X 0,Y 148.124,Z 381.056,A -85,B 0,C 180,E1 -24034.87,E2 -24034.87} C_VEL
LIN {X 0,Y 148.687,Z 379.923,A -85,B 0,C 180,E1 -24038.153,E2 -24038.153} C_VEL
LIN {X 0,Y 149.336,Z 378.571,A -85,B 0,C 180,E1 -24040.852,E2 -24040.852} C_VEL
LIN {X 0,Y 150.801,Z 375.709,A -85,B 0,C 180,E1 -24044.853,E2 -24044.853} C_VEL
LIN {X 0,Y 152.939,Z 371.822,A -85,B 0,C 180,E1 -24048.765,E2 -24048.765} C_VEL
LIN {X 0,Y 155.66,Z 366.806,A -85,B 0,C 180,E1 -24052.569,E2 -24052.569} C_VEL
LIN {X 0,Y 159.012,Z 360.483,A -85,B 0,C 180,E1 -24056.231,E2 -24056.231} C_VEL
LIN {X 0,Y 162.963,Z 352.568,A -85,B 0,C 180,E1 -24059.734,E2 -24059.734} C_VEL
LIN {X 0,Y 166.454,Z 344.542,A -85,B 0,C 180,E1 -24062.556,E2 -24062.556} C_VEL
LIN {X 0,Y 170.385,Z 334.658,A -85,B 0,C 180,E1 -24065.274,E2 -24065.274} C_VEL
LIN {X 0,Y 174.289,Z 323.558,A -85,B 0,C 180,E1 -24067.583,E2 -24067.583} C_VEL
LIN {X 0,Y 177.449,Z 312.675,A -85,B 0,C 180,E1 -24069.324,E2 -24069.324} C_VEL
LIN {X 0,Y 180.255,Z 300.64,A -85,B 0,C 180,E1 -24070.774,E2 -24070.774} C_VEL
LIN {X 0,Y 182.365,Z 288.102,A -85,B 0,C 180,E1 -24071.864,E2 -24071.864} C_VEL
LIN {X 0,Y 183.831,Z 274.91,A -85,B 0,C 180,E1 -24072.571,E2 -24072.571} C_VEL
LIN {X 0,Y 186.227,Z 235.185,A -85,B 0,C 180,E1 -24073.976,E2 -24073.976} C_VEL
LIN {X 0,Y 181.737,Z 225.894,A -85,B 0,C 180,E1 -24075.886,E2 -24075.886} C_VEL
LIN {X 0,Y 175.88,Z 215.63,A -85,B 0,C 180,E1 -24078.527,E2 -24078.527} C_VEL
LIN {X 0,Y 170.226,Z 206.843,A -85,B 0,C 180,E1 -24081.328,E2 -24081.328} C_VEL
LIN {X 0,Y 165.184,Z 199.578,A -85,B 0,C 180,E1 -24084.116,E2 -24084.116} C_VEL
LIN {X 0,Y 161.905,Z 195.118,A -85,B 0,C 180,E1 -24086.115,E2 -24086.115} C_VEL
LIN {X 0,Y 159.274,Z 191.703,A -85,B 0,C 180,E1 -24087.848,E2 -24087.848} C_VEL
LIN {X 0,Y 158.475,Z 190.573,A -85,B 0,C 180,E1 -24088.412,E2 -24088.412} C_VEL
LIN {X 0,Y 155.947,Z 187.925,A -85,B 0,C 180,E1 -24090.212,E2 -24090.212} C_VEL
LIN {X 0,Y 154.639,Z 185.476,A -85,B 0,C 180,E1 -24091.312,E2 -24091.312} C_VEL
LIN {X 0,Y 152.274,Z 183.864,A -85,B 0,C 180,E1 -24093.165,E2 -24093.165} C_VEL
LIN {X 0,Y 150.731,Z 181.674,A -85,B 0,C 180,E1 -24094.601,E2 -24094.601} C_VEL
LIN {X 0,Y 150.236,Z 179.759,A -85,B 0,C 180,E1 -24095.286,E2 -24095.286} C_VEL
LIN {X 0,Y 150.301,Z 179.764,A -85,B 0,C 180,E1 -24100.894,E2 -24100.894} C_VEL
LIN {X 0,Y 150.405,Z 179.727,A -85,B 0,C 180,E1 -24106.489,E2 -24106.489} C_VEL
LIN {X 0,Y 150.607,Z 179.725,A -85,B 0,C 180,E1 -24109.242,E2 -24109.242} C_VEL
LIN {X 0,Y 150.681,Z 179.687,A -85,B 0,C 180,E1 -24111.956,E2 -24111.956} C_VEL
LIN {X 0,Y 151.196,Z 179.623,A -85,B 0,C 180,E1 -24120,E2 -24120} C_VEL
LIN {X 0,Y 150.677,Z 179.69,A -85,B 0,C 180,E1 -24128.044,E2 -24128.044} C_VEL
LIN {X 0,Y 150.57,Z 179.711,A -85,B 0,C 180,E1 -24131.42,E2 -24131.42} C_VEL
LIN {X 0,Y 150.304,Z 179.735,A -85,B 0,C 180,E1 -24136.293,E2 -24136.293} C_VEL
LIN {X 0,Y 150.283,Z 179.761,A -85,B 0,C 180,E1 -24140.721,E2 -24140.721} C_VEL
LIN {X 0,Y 150.212,Z 179.755,A -85,B 0,C 180,E1 -24144.258,E2 -24144.258} C_VEL
LIN {X 0,Y 150.896,Z 182.056,A -85,B 0,C 180,E1 -24145.105,E2 -24145.105} C_VEL
LIN {X 0,Y 152.597,Z 184.241,A -85,B 0,C 180,E1 -24146.646,E2 -24146.646} C_VEL
LIN {X 0,Y 154.73,Z 185.658,A -85,B 0,C 180,E1 -24148.299,E2 -24148.299} C_VEL
LIN {X 0,Y 156.498,Z 188.707,A -85,B 0,C 180,E1 -24149.743,E2 -24149.743} C_VEL
LIN {X 0,Y 159.008,Z 191.238,A -85,B 0,C 180,E1 -24151.489,E2 -24151.489} C_VEL
LIN {X 0,Y 161.465,Z 194.696,A -85,B 0,C 180,E1 -24153.148,E2 -24153.148} C_VEL
LIN {X 0,Y 162.991,Z 196.529,A -85,B 0,C 180,E1 -24154.094,E2 -24154.094} C_VEL
LIN {X 0,Y 168.879,Z 206.257,A -85,B 0,C 180,E1 -24157.584,E2 -24157.584} C_VEL
LIN {X 0,Y 173.83,Z 215.623,A -85,B 0,C 180,E1 -24160.227,E2 -24160.227} C_VEL
LIN {X 0,Y 178.607,Z 225.375,A -85,B 0,C 180,E1 -24162.561,E2 -24162.561} C_VEL
LIN {X 0,Y 184.066,Z 238.951,A -85,B 0,C 180,E1 -24165.1,E2 -24165.1} C_VEL
LIN {X 0,Y 185.18,Z 242.335,A -85,B 0,C 180,E1 -24165.619,E2 -24165.619} C_VEL
LIN {X 0,Y 185.512,Z 248.219,A -85,B 0,C 180,E1 -24166.028,E2 -24166.028} C_VEL
LIN {X 0,Y 182.892,Z 288.619,A -85,B 0,C 180,E1 -24167.467,E2 -24167.467} C_VEL
LIN {X 0,Y 181.026,Z 302.168,A -85,B 0,C 180,E1 -24168.301,E2 -24168.301} C_VEL
LIN {X 0,Y 178.384,Z 314.788,A -85,B 0,C 180,E1 -24169.452,E2 -24169.452} C_VEL
LIN {X 0,Y 174.86,Z 327.447,A -85,B 0,C 180,E1 -24171.096,E2 -24171.096} C_VEL
LIN {X 0,Y 171.122,Z 338.716,A -85,B 0,C 180,E1 -24173.083,E2 -24173.083} C_VEL
LIN {X 0,Y 167.184,Z 348.868,A -85,B 0,C 180,E1 -24175.423,E2 -24175.423} C_VEL
LIN {X 0,Y 163.194,Z 358.021,A -85,B 0,C 180,E1 -24178.159,E2 -24178.159} C_VEL
LIN {X 0,Y 159.028,Z 367.091,A -85,B 0,C 180,E1 -24181.706,E2 -24181.706} C_VEL
LIN {X 0,Y 155.647,Z 374.171,A -85,B 0,C 180,E1 -24185.325,E2 -24185.325} C_VEL
LIN {X 0,Y 153.101,Z 379.006,A -85,B 0,C 180,E1 -24188.454,E2 -24188.454} C_VEL
LIN {X 0,Y 150.67,Z 383.73,A -85,B 0,C 180,E1 -24192.349,E2 -24192.349} C_VEL
LIN {X 0,Y 149.451,Z 386.384,A -85,B 0,C 180,E1 -24195.157,E2 -24195.157} C_VEL
LIN {X 0,Y 148.096,Z 388.047,A -85,B 0,C 180,E1 -24197.284,E2 -24197.284} C_VEL
LIN {X 0,Y 144.421,Z 390.148,A -85,B 0,C 180,E1 -24200.803,E2 -24200.803} C_VEL
LIN {X 0,Y 141.674,Z 391.254,A -85,B 0,C 180,E1 -24203.767,E2 -24203.767} C_VEL
LIN {X 0,Y 140.614,Z 391.815,A -85,B 0,C 180,E1 -24206.124,E2 -24206.124} C_VEL
LIN {X 0,Y 140.572,Z 391.944,A -85,B 0,C 180,E1 -24206.926,E2 -24206.926} C_VEL
LIN {X 0,Y 140.69,Z 392.205,A -85,B 0,C 180,E1 -24209.998,E2 -24209.998} C_VEL
LIN {X 0,Y 140.547,Z 391.971,A -85,B 0,C 180,E1 -24212.865,E2 -24212.865} C_VEL
LIN {X 0,Y 140.609,Z 391.346,A -85,B 0,C 180,E1 -24215.736,E2 -24215.736} C_VEL
LIN {X 0,Y 141.339,Z 388.909,A -85,B 0,C 180,E1 -24221.471,E2 -24221.471} C_VEL
LIN {X 0,Y 142.611,Z 385.939,A -85,B 0,C 180,E1 -24225.725,E2 -24225.725} C_VEL
LIN {X 0,Y 144.687,Z 381.936,A -85,B 0,C 180,E1 -24229.876,E2 -24229.876} C_VEL
LIN {X 0,Y 148.044,Z 375.791,A -85,B 0,C 180,E1 -24234.542,E2 -24234.542} C_VEL
LIN {X 0,Y 151.51,Z 369.085,A -85,B 0,C 180,E1 -24238.387,E2 -24238.387} C_VEL
LIN {X 0,Y 155.639,Z 360.773,A -85,B 0,C 180,E1 -24242.043,E2 -24242.043} C_VEL
LIN {X 0,Y 159.622,Z 352.255,A -85,B 0,C 180,E1 -24244.914,E2 -24244.914} C_VEL
LIN {X 0,Y 164.091,Z 341.739,A -85,B 0,C 180,E1 -24247.611,E2 -24247.611} C_VEL
LIN {X 0,Y 167.87,Z 331.332,A -85,B 0,C 180,E1 -24249.674,E2 -24249.674} C_VEL
LIN {X 0,Y 171.457,Z 319.917,A -85,B 0,C 180,E1 -24251.371,E2 -24251.371} C_VEL
LIN {X 0,Y 174.37,Z 308.147,A -85,B 0,C 180,E1 -24252.656,E2 -24252.656} C_VEL
LIN {X 0,Y 176.76,Z 294.685,A -85,B 0,C 180,E1 -24253.681,E2 -24253.681} C_VEL
LIN {X 0,Y 178.047,Z 281.806,A -85,B 0,C 180,E1 -24254.322,E2 -24254.322} C_VEL
LIN {X 0,Y 180.273,Z 247.713,A -85,B 0,C 180,E1 -24255.501,E2 -24255.501} C_VEL
LIN {X 0,Y 179.774,Z 243.735,A -85,B 0,C 180,E1 -24255.883,E2 -24255.883} C_VEL
LIN {X 0,Y 175.048,Z 231.359,A -85,B 0,C 180,E1 -24258.224,E2 -24258.224} C_VEL
LIN {X 0,Y 170.698,Z 221.877,A -85,B 0,C 180,E1 -24260.475,E2 -24260.475} C_VEL
LIN {X 0,Y 165.589,Z 211.9,A -85,B 0,C 180,E1 -24263.346,E2 -24263.346} C_VEL
LIN {X 0,Y 161.215,Z 204.397,A -85,B 0,C 180,E1 -24266.045,E2 -24266.045} C_VEL
LIN {X 0,Y 159.239,Z 201.169,A -85,B 0,C 180,E1 -24267.366,E2 -24267.366} C_VEL
LIN {X 0,Y 156.512,Z 197.512,A -85,B 0,C 180,E1 -24269.259,E2 -24269.259} C_VEL
LIN {X 0,Y 153.024,Z 193.224,A -85,B 0,C 180,E1 -24271.917,E2 -24271.917} C_VEL
LIN {X 0,Y 152.107,Z 191.828,A -85,B 0,C 180,E1 -24272.703,E2 -24272.703} C_VEL
LIN {X 0,Y 149.478,Z 189.39,A -85,B 0,C 180,E1 -24274.966,E2 -24274.966} C_VEL
LIN {X 0,Y 147.98,Z 186.488,A -85,B 0,C 180,E1 -24276.562,E2 -24276.562} C_VEL
LIN {X 0,Y 145.552,Z 185.066,A -85,B 0,C 180,E1 -24279.031,E2 -24279.031} C_VEL
LIN {X 0,Y 143.78,Z 182.636,A -85,B 0,C 180,E1 -24281.29,E2 -24281.29} C_VEL
LIN {X 0,Y 143.213,Z 180.627,A -85,B 0,C 180,E1 -24282.323,E2 -24282.323} C_VEL
LIN {X 0,Y 143.525,Z 180.589,A -85,B 0,C 180,E1 -24288.705,E2 -24288.705} C_VEL
LIN {X 0,Y 143.597,Z 180.578,A -85,B 0,C 180,E1 -24291.557,E2 -24291.557} C_VEL
LIN {X 0,Y 144.147,Z 180.52,A -85,B 0,C 180,E1 -24300,E2 -24300} C_VEL
LIN {X 0,Y 143.612,Z 180.596,A -85,B 0,C 180,E1 -24308.442,E2 -24308.442} C_VEL
LIN {X 0,Y 143.489,Z 180.587,A -85,B 0,C 180,E1 -24311.608,E2 -24311.608} C_VEL
LIN {X 0,Y 143.235,Z 180.696,A -85,B 0,C 180,E1 -24318.321,E2 -24318.321} C_VEL
LIN {X 0,Y 144.013,Z 183.087,A -85,B 0,C 180,E1 -24319.604,E2 -24319.604} C_VEL
LIN {X 0,Y 145.98,Z 185.459,A -85,B 0,C 180,E1 -24322.007,E2 -24322.007} C_VEL
LIN {X 0,Y 148.12,Z 186.807,A -85,B 0,C 180,E1 -24324.157,E2 -24324.157} C_VEL
LIN {X 0,Y 149.921,Z 189.942,A -85,B 0,C 180,E1 -24326.008,E2 -24326.008} C_VEL
LIN {X 0,Y 152.601,Z 192.364,A -85,B 0,C 180,E1 -24328.262,E2 -24328.262} C_VEL
LIN {X 0,Y 154.913,Z 195.809,A -85,B 0,C 180,E1 -24330.147,E2 -24330.147} C_VEL
LIN {X 0,Y 156.628,Z 197.678,A -85,B 0,C 180,E1 -24331.385,E2 -24331.385} C_VEL
LIN {X 0,Y 159.352,Z 201.303,A -85,B 0,C 180,E1 -24333.267,E2 -24333.267} C_VEL
LIN {X 0,Y 164.218,Z 208.321,A -85,B 0,C 180,E1 -24336.312,E2 -24336.312} C_VEL
LIN {X 0,Y 169.97,Z 217.076,A -85,B 0,C 180,E1 -24339.475,E2 -24339.475} C_VEL
LIN {X 0,Y 175.905,Z 227.427,A -85,B 0,C 180,E1 -24342.41,E2 -24342.41} C_VEL
LIN {X 0,Y 180.884,Z 237.309,A -85,B 0,C 180,E1 -24344.677,E2 -24344.677} C_VEL
LIN {X 0,Y 178.657,Z 272.704,A -85,B 0,C 180,E1 -24345.929,E2 -24345.929} C_VEL
LIN {X 0,Y 177.319,Z 285.727,A -85,B 0,C 180,E1 -24346.581,E2 -24346.581} C_VEL
LIN {X 0,Y 175.219,Z 298.441,A -85,B 0,C 180,E1 -24347.599,E2 -24347.599} C_VEL
LIN {X 0,Y 172.542,Z 310.257,A -85,B 0,C 180,E1 -24348.946,E2 -24348.946} C_VEL
LIN {X 0,Y 169.254,Z 321.665,A -85,B 0,C 180,E1 -24350.713,E2 -24350.713} C_VEL
LIN {X 0,Y 165.108,Z 333.211,A -85,B 0,C 180,E1 -24353.043,E2 -24353.043} C_VEL
LIN {X 0,Y 161.387,Z 342.505,A -85,B 0,C 180,E1 -24355.522,E2 -24355.522} C_VEL
LIN {X 0,Y 157.636,Z 350.965,A -85,B 0,C 180,E1 -24358.411,E2 -24358.411} C_VEL
LIN {X 0,Y 153.444,Z 359.197,A -85,B 0,C 180,E1 -24362.002,E2 -24362.002} C_VEL
LIN {X 0,Y 150.277,Z 364.829,A -85,B 0,C 180,E1 -24365.11,E2 -24365.11} C_VEL
LIN {X 0,Y 147.192,Z 370.311,A -85,B 0,C 180,E1 -24369.018,E2 -24369.018} C_VEL
LIN {X 0,Y 144.695,Z 374.611,A -85,B 0,C 180,E1 -24373.058,E2 -24373.058} C_VEL
LIN {X 0,Y 143.387,Z 376.884,A -85,B 0,C 180,E1 -24375.816,E2 -24375.816} C_VEL
LIN {X 0,Y 142.366,Z 378.73,A -85,B 0,C 180,E1 -24378.613,E2 -24378.613} C_VEL
LIN {X 0,Y 141.667,Z 380.113,A -85,B 0,C 180,E1 -24381.443,E2 -24381.443} C_VEL
LIN {X 0,Y 140.865,Z 381.702,A -85,B 0,C 180,E1 -24387.142,E2 -24387.142} C_VEL
LIN {X 0,Y 140.818,Z 381.926,A -85,B 0,C 180,E1 -24390.002,E2 -24390.002} C_VEL
LIN {X 0,Y 141.01,Z 381.447,A -85,B 0,C 180,E1 -24394.576,E2 -24394.576} C_VEL
LIN {X 0,Y 141.667,Z 380.182,A -85,B 0,C 180,E1 -24398.56,E2 -24398.56} C_VEL
LIN {X 0,Y 142.356,Z 378.83,A -85,B 0,C 180,E1 -24401.391,E2 -24401.391} C_VEL
LIN {X 0,Y 143.964,Z 375.967,A -85,B 0,C 180,E1 -24405.576,E2 -24405.576} C_VEL
LIN {X 0,Y 146.229,Z 372.081,A -85,B 0,C 180,E1 -24409.661,E2 -24409.661} C_VEL
LIN {X 0,Y 149.119,Z 367.064,A -85,B 0,C 180,E1 -24413.617,E2 -24413.617} C_VEL
LIN {X 0,Y 152.682,Z 360.74,A -85,B 0,C 180,E1 -24417.408,E2 -24417.408} C_VEL
LIN {X 0,Y 156.839,Z 352.825,A -85,B 0,C 180,E1 -24421.02,E2 -24421.02} C_VEL
LIN {X 0,Y 160.861,Z 344.022,A -85,B 0,C 180,E1 -24424.167,E2 -24424.167} C_VEL
LIN {X 0,Y 164.646,Z 334.914,A -85,B 0,C 180,E1 -24426.699,E2 -24426.699} C_VEL
LIN {X 0,Y 168.732,Z 323.812,A -85,B 0,C 180,E1 -24429.05,E2 -24429.05} C_VEL
LIN {X 0,Y 172.03,Z 312.928,A -85,B 0,C 180,E1 -24430.818,E2 -24430.818} C_VEL
LIN {X 0,Y 174.958,Z 300.891,A -85,B 0,C 180,E1 -24432.288,E2 -24432.288} C_VEL
LIN {X 0,Y 177.141,Z 288.476,A -85,B 0,C 180,E1 -24433.383,E2 -24433.383} C_VEL
LIN {X 0,Y 178.685,Z 275.113,A -85,B 0,C 180,E1 -24434.108,E2 -24434.108} C_VEL
LIN {X 0,Y 181.05,Z 237.535,A -85,B 0,C 180,E1 -24435.461,E2 -24435.461} C_VEL
LIN {X 0,Y 176.309,Z 227.982,A -85,B 0,C 180,E1 -24437.628,E2 -24437.628} C_VEL
LIN {X 0,Y 169.896,Z 216.833,A -85,B 0,C 180,E1 -24440.805,E2 -24440.805} C_VEL
LIN {X 0,Y 164.104,Z 208.1,A -85,B 0,C 180,E1 -24444.015,E2 -24444.015} C_VEL
LIN {X 0,Y 161.686,Z 204.663,A -85,B 0,C 180,E1 -24445.487,E2 -24445.487} C_VEL
LIN {X 0,Y 158.894,Z 200.76,A -85,B 0,C 180,E1 -24447.314,E2 -24447.314} C_VEL
LIN {X 0,Y 155.916,Z 196.718,A -85,B 0,C 180,E1 -24449.437,E2 -24449.437} C_VEL
LIN {X 0,Y 153.249,Z 193.533,A -85,B 0,C 180,E1 -24451.495,E2 -24451.495} C_VEL
LIN {X 0,Y 152.259,Z 191.895,A -85,B 0,C 180,E1 -24452.36,E2 -24452.36} C_VEL
LIN {X 0,Y 149.772,Z 189.726,A -85,B 0,C 180,E1 -24454.493,E2 -24454.493} C_VEL
LIN {X 0,Y 148.206,Z 186.932,A -85,B 0,C 180,E1 -24456.136,E2 -24456.136} C_VEL
LIN {X 0,Y 147.826,Z 186.424,A -85,B 0,C 180,E1 -24456.536,E2 -24456.536} C_VEL
LIN {X 0,Y 145.286,Z 184.794,A -85,B 0,C 180,E1 -24459.218,E2 -24459.218} C_VEL
LIN {X 0,Y 143.627,Z 182.252,A -85,B 0,C 180,E1 -24461.454,E2 -24461.454} C_VEL
LIN {X 0,Y 143.224,Z 180.632,A -85,B 0,C 180,E1 -24462.325,E2 -24462.325} C_VEL
LIN {X 0,Y 143.534,Z 180.606,A -85,B 0,C 180,E1 -24468.705,E2 -24468.705} C_VEL
LIN {X 0,Y 143.607,Z 180.569,A -85,B 0,C 180,E1 -24471.557,E2 -24471.557} C_VEL
LIN {X 0,Y 144.154,Z 180.499,A -85,B 0,C 180,E1 -24480,E2 -24480} C_VEL
LIN {X 0,Y 143.603,Z 180.567,A -85,B 0,C 180,E1 -24488.443,E2 -24488.443} C_VEL
LIN {X 0,Y 143.495,Z 180.593,A -85,B 0,C 180,E1 -24491.604,E2 -24491.604} C_VEL
LIN {X 0,Y 143.26,Z 180.796,A -85,B 0,C 180,E1 -24497.394,E2 -24497.394} C_VEL
LIN {X 0,Y 143.793,Z 182.661,A -85,B 0,C 180,E1 -24498.339,E2 -24498.339} C_VEL
LIN {X 0,Y 145.636,Z 185.131,A -85,B 0,C 180,E1 -24500.724,E2 -24500.724} C_VEL
LIN {X 0,Y 148.065,Z 186.659,A -85,B 0,C 180,E1 -24503.238,E2 -24503.238} C_VEL
LIN {X 0,Y 149.549,Z 189.537,A -85,B 0,C 180,E1 -24504.836,E2 -24504.836} C_VEL
LIN {X 0,Y 152.558,Z 192.33,A -85,B 0,C 180,E1 -24507.431,E2 -24507.431} C_VEL
LIN {X 0,Y 154.924,Z 195.768,A -85,B 0,C 180,E1 -24509.374,E2 -24509.374} C_VEL
LIN {X 0,Y 156.478,Z 197.401,A -85,B 0,C 180,E1 -24510.504,E2 -24510.504} C_VEL
LIN {X 0,Y 159.136,Z 201.039,A -85,B 0,C 180,E1 -24512.377,E2 -24512.377} C_VEL
LIN {X 0,Y 160.493,Z 202.98,A -85,B 0,C 180,E1 -24513.281,E2 -24513.281} C_VEL
LIN {X 0,Y 165.779,Z 212.076,A -85,B 0,C 180,E1 -24516.596,E2 -24516.596} C_VEL
LIN {X 0,Y 170.926,Z 222.186,A -85,B 0,C 180,E1 -24519.497,E2 -24519.497} C_VEL
LIN {X 0,Y 174.831,Z 230.73,A -85,B 0,C 180,E1 -24521.531,E2 -24521.531} C_VEL
LIN {X 0,Y 179.613,Z 242.935,A -85,B 0,C 180,E1 -24523.903,E2 -24523.903} C_VEL
LIN {X 0,Y 180.284,Z 245.572,A -85,B 0,C 180,E1 -24524.269,E2 -24524.269} C_VEL
LIN {X 0,Y 180.375,Z 249.496,A -85,B 0,C 180,E1 -24524.516,E2 -24524.516} C_VEL
LIN {X 0,Y 177.672,Z 288.793,A -85,B 0,C 180,E1 -24525.939,E2 -24525.939} C_VEL
LIN {X 0,Y 175.755,Z 302.146,A -85,B 0,C 180,E1 -24526.781,E2 -24526.781} C_VEL
LIN {X 0,Y 173.064,Z 314.536,A -85,B 0,C 180,E1 -24527.928,E2 -24527.928} C_VEL
LIN {X 0,Y 169.917,Z 325.609,A -85,B 0,C 180,E1 -24529.349,E2 -24529.349} C_VEL
LIN {X 0,Y 165.949,Z 337.165,A -85,B 0,C 180,E1 -24531.341,E2 -24531.341} C_VEL
LIN {X 0,Y 161.825,Z 347.578,A -85,B 0,C 180,E1 -24533.719,E2 -24533.719} C_VEL
LIN {X 0,Y 158.001,Z 356.095,A -85,B 0,C 180,E1 -24536.219,E2 -24536.219} C_VEL
LIN {X 0,Y 154.198,Z 363.959,A -85,B 0,C 180,E1 -24539.152,E2 -24539.152} C_VEL
LIN {X 0,Y 150.186,Z 371.804,A -85,B 0,C 180,E1 -24542.959,E2 -24542.959} C_VEL
LIN {X 0,Y 147.472,Z 376.921,A -85,B 0,C 180,E1 -24546.103,E2 -24546.103} C_VEL
LIN {X 0,Y 144.69,Z 382.033,A -85,B 0,C 180,E1 -24550.121,E2 -24550.121} C_VEL
LIN {X 0,Y 142.431,Z 386.398,A -85,B 0,C 180,E1 -24554.779,E2 -24554.779} C_VEL
LIN {X 0,Y 141.335,Z 388.958,A -85,B 0,C 180,E1 -24558.526,E2 -24558.526} C_VEL
LIN {X 0,Y 140.548,Z 391.369,A -85,B 0,C 180,E1 -24564.259,E2 -24564.259} C_VEL
LIN {X 0,Y 140.572,Z 391.944,A -85,B 0,C 180,E1 -24566.926,E2 -24566.926} C_VEL
LIN {X 0,Y 140.324,Z 392.194,A -85,B 0,C 180,E1 -24568.52,E2 -24568.52} C_VEL
LIN {X 0,Y 139.531,Z 392.268,A -85,B 0,C 180,E1 -24570.099,E2 -24570.099} C_VEL
LIN {X 0,Y 137.1,Z 391.951,A -85,B 0,C 180,E1 -24573.235,E2 -24573.235} C_VEL
LIN {X 0,Y 134.71,Z 391.073,A -85,B 0,C 180,E1 -24576.476,E2 -24576.476} C_VEL
LIN {X 0,Y 133.87,Z 390.099,A -85,B 0,C 180,E1 -24578.988,E2 -24578.988} C_VEL
LIN {X 0,Y 133.902,Z 389.708,A -85,B 0,C 180,E1 -24579.832,E2 -24579.832} C_VEL
LIN {X 0,Y 135.223,Z 386.76,A -85,B 0,C 180,E1 -24585.06,E2 -24585.06} C_VEL
LIN {X 0,Y 137.152,Z 383.112,A -85,B 0,C 180,E1 -24589.454,E2 -24589.454} C_VEL
LIN {X 0,Y 139.892,Z 378.36,A -85,B 0,C 180,E1 -24593.696,E2 -24593.696} C_VEL
LIN {X 0,Y 143.672,Z 371.786,A -85,B 0,C 180,E1 -24598.093,E2 -24598.093} C_VEL
LIN {X 0,Y 147.371,Z 364.887,A -85,B 0,C 180,E1 -24601.638,E2 -24601.638} C_VEL
LIN {X 0,Y 151.285,Z 357.28,A -85,B 0,C 180,E1 -24604.684,E2 -24604.684} C_VEL
LIN {X 0,Y 155.669,Z 348.075,A -85,B 0,C 180,E1 -24607.55,E2 -24607.55} C_VEL
LIN {X 0,Y 159.944,Z 337.84,A -85,B 0,C 180,E1 -24609.986,E2 -24609.986} C_VEL
LIN {X 0,Y 164.034,Z 326.494,A -85,B 0,C 180,E1 -24612.022,E2 -24612.022} C_VEL
LIN {X 0,Y 167.563,Z 314.715,A -85,B 0,C 180,E1 -24613.582,E2 -24613.582} C_VEL
LIN {X 0,Y 170.462,Z 301.793,A -85,B 0,C 180,E1 -24614.805,E2 -24614.805} C_VEL
LIN {X 0,Y 172.498,Z 288.118,A -85,B 0,C 180,E1 -24615.665,E2 -24615.665} C_VEL
LIN {X 0,Y 175.271,Z 248.559,A -85,B 0,C 180,E1 -24617.124,E2 -24617.124} C_VEL
LIN {X 0,Y 174.877,Z 246.277,A -85,B 0,C 180,E1 -24617.396,E2 -24617.396} C_VEL
LIN {X 0,Y 170.061,Z 233.499,A -85,B 0,C 180,E1 -24619.984,E2 -24619.984} C_VEL
LIN {X 0,Y 164.935,Z 222.477,A -85,B 0,C 180,E1 -24622.9,E2 -24622.9} C_VEL
LIN {X 0,Y 160.811,Z 214.508,A -85,B 0,C 180,E1 -24625.474,E2 -24625.474} C_VEL
LIN {X 0,Y 156.645,Z 207.233,A -85,B 0,C 180,E1 -24628.343,E2 -24628.343} C_VEL
LIN {X 0,Y 153.861,Z 203.331,A -85,B 0,C 180,E1 -24630.404,E2 -24630.404} C_VEL
LIN {X 0,Y 150.684,Z 199.343,A -85,B 0,C 180,E1 -24632.982,E2 -24632.982} C_VEL
LIN {X 0,Y 149.98,Z 198.299,A -85,B 0,C 180,E1 -24633.617,E2 -24633.617} C_VEL
LIN {X 0,Y 147.168,Z 195.284,A -85,B 0,C 180,E1 -24636.238,E2 -24636.238} C_VEL
LIN {X 0,Y 145.895,Z 193.105,A -85,B 0,C 180,E1 -24637.657,E2 -24637.657} C_VEL
LIN {X 0,Y 143.251,Z 190.943,A -85,B 0,C 180,E1 -24640.661,E2 -24640.661} C_VEL
LIN {X 0,Y 141.657,Z 187.945,A -85,B 0,C 180,E1 -24643.054,E2 -24643.054} C_VEL
LIN {X 0,Y 141.452,Z 187.496,A -85,B 0,C 180,E1 -24643.4,E2 -24643.4} C_VEL
LIN {X 0,Y 138.733,Z 185.92,A -85,B 0,C 180,E1 -24647.985,E2 -24647.985} C_VEL
LIN {X 0,Y 136.667,Z 182.206,A -85,B 0,C 180,E1 -24654.652,E2 -24654.652} C_VEL
LIN {X 0,Y 136.579,Z 181.452,A -85,B 0,C 180,E1 -24655.758,E2 -24655.758} C_VEL
LIN {X 0,Y 137.104,Z 181.396,A -85,B 0,C 180,E1 -24660,E2 -24660} C_VEL
LIN {X 0,Y 136.557,Z 181.475,A -85,B 0,C 180,E1 -24664.982,E2 -24664.982} C_VEL
LIN {X 0,Y 137.124,Z 183.514,A -85,B 0,C 180,E1 -24668.103,E2 -24668.103} C_VEL
LIN {X 0,Y 139.764,Z 186.795,A -85,B 0,C 180,E1 -24674.562,E2 -24674.562} C_VEL
LIN {X 0,Y 141.616,Z 187.741,A -85,B 0,C 180,E1 -24677.417,E2 -24677.417} C_VEL
LIN {X 0,Y 142.997,Z 190.613,A -85,B 0,C 180,E1 -24679.562,E2 -24679.562} C_VEL
LIN {X 0,Y 145.373,Z 192.847,A -85,B 0,C 180,E1 -24682.37,E2 -24682.37} C_VEL
LIN {X 0,Y 146.232,Z 193.505,A -85,B 0,C 180,E1 -24683.266,E2 -24683.266} C_VEL
LIN {X 0,Y 148.454,Z 196.946,A -85,B 0,C 180,E1 -24685.594,E2 -24685.594} C_VEL
LIN {X 0,Y 150.469,Z 198.906,A -85,B 0,C 180,E1 -24687.373,E2 -24687.373} C_VEL
LIN {X 0,Y 153.085,Z 202.552,A -85,B 0,C 180,E1 -24689.573,E2 -24689.573} C_VEL
LIN {X 0,Y 154.396,Z 204.219,A -85,B 0,C 180,E1 -24690.579,E2 -24690.579} C_VEL
LIN {X 0,Y 157.736,Z 208.913,A -85,B 0,C 180,E1 -24692.985,E2 -24692.985} C_VEL
LIN {X 0,Y 162.201,Z 215.416,A -85,B 0,C 180,E1 -24695.852,E2 -24695.852} C_VEL
LIN {X 0,Y 167.984,Z 224.872,A -85,B 0,C 180,E1 -24699.16,E2 -24699.16} C_VEL
LIN {X 0,Y 173.85,Z 235.734,A -85,B 0,C 180,E1 -24702.162,E2 -24702.162} C_VEL
LIN {X 0,Y 175.822,Z 239.95,A -85,B 0,C 180,E1 -24703.122,E2 -24703.122} C_VEL
LIN {X 0,Y 173.194,Z 278.315,A -85,B 0,C 180,E1 -24704.528,E2 -24704.528} C_VEL
LIN {X 0,Y 171.407,Z 291.385,A -85,B 0,C 180,E1 -24705.344,E2 -24705.344} C_VEL
LIN {X 0,Y 168.772,Z 304.508,A -85,B 0,C 180,E1 -24706.602,E2 -24706.602} C_VEL
LIN {X 0,Y 165.857,Z 315.777,A -85,B 0,C 180,E1 -24708.137,E2 -24708.137} C_VEL
LIN {X 0,Y 161.875,Z 327.393,A -85,B 0,C 180,E1 -24710.182,E2 -24710.182} C_VEL
LIN {X 0,Y 157.734,Z 337.822,A -85,B 0,C 180,E1 -24712.624,E2 -24712.624} C_VEL
LIN {X 0,Y 153.752,Z 346.801,A -85,B 0,C 180,E1 -24715.365,E2 -24715.365} C_VEL
LIN {X 0,Y 149.344,Z 355.563,A -85,B 0,C 180,E1 -24718.827,E2 -24718.827} C_VEL
LIN {X 0,Y 145.156,Z 362.957,A -85,B 0,C 180,E1 -24722.618,E2 -24722.618} C_VEL
LIN {X 0,Y 141.611,Z 368.885,A -85,B 0,C 180,E1 -24726.609,E2 -24726.609} C_VEL
LIN {X 0,Y 138.716,Z 373.567,A -85,B 0,C 180,E1 -24730.774,E2 -24730.774} C_VEL
LIN {X 0,Y 136.521,Z 377.144,A -85,B 0,C 180,E1 -24735.086,E2 -24735.086} C_VEL
LIN {X 0,Y 135.404,Z 378.99,A -85,B 0,C 180,E1 -24738.019,E2 -24738.019} C_VEL
LIN {X 0,Y 134.646,Z 380.372,A -85,B 0,C 180,E1 -24740.993,E2 -24740.993} C_VEL
LIN {X 0,Y 133.786,Z 381.961,A -85,B 0,C 180,E1 -24746.99,E2 -24746.99} C_VEL
LIN {X 0,Y 133.722,Z 382.185,A -85,B 0,C 180,E1 -24750.002,E2 -24750.002} C_VEL
LIN {X 0,Y 133.858,Z 381.836,A -85,B 0,C 180,E1 -24753.995,E2 -24753.995} C_VEL
LIN {X 0,Y 134.646,Z 380.441,A -85,B 0,C 180,E1 -24759.01,E2 -24759.01} C_VEL
LIN {X 0,Y 135.393,Z 379.089,A -85,B 0,C 180,E1 -24761.985,E2 -24761.985} C_VEL
LIN {X 0,Y 137.129,Z 376.226,A -85,B 0,C 180,E1 -24766.374,E2 -24766.374} C_VEL
LIN {X 0,Y 139.566,Z 372.339,A -85,B 0,C 180,E1 -24770.641,E2 -24770.641} C_VEL
LIN {X 0,Y 142.639,Z 367.322,A -85,B 0,C 180,E1 -24774.76,E2 -24774.76} C_VEL
LIN {X 0,Y 146.422,Z 360.997,A -85,B 0,C 180,E1 -24778.685,E2 -24778.685} C_VEL
LIN {X 0,Y 150.783,Z 353.082,A -85,B 0,C 180,E1 -24782.414,E2 -24782.414} C_VEL
LIN {X 0,Y 154.72,Z 344.987,A -85,B 0,C 180,E1 -24785.406,E2 -24785.406} C_VEL
LIN {X 0,Y 159.008,Z 335.169,A -85,B 0,C 180,E1 -24788.229,E2 -24788.229} C_VEL
LIN {X 0,Y 163.277,Z 324.066,A -85,B 0,C 180,E1 -24790.62,E2 -24790.62} C_VEL
LIN {X 0,Y 166.724,Z 313.181,A -85,B 0,C 180,E1 -24792.413,E2 -24792.413} C_VEL
LIN {X 0,Y 169.5,Z 302.27,A -85,B 0,C 180,E1 -24793.783,E2 -24793.783} C_VEL
LIN {X 0,Y 171.981,Z 289.377,A -85,B 0,C 180,E1 -24794.95,E2 -24794.95} C_VEL
LIN {X 0,Y 173.564,Z 276.575,A -85,B 0,C 180,E1 -24795.686,E2 -24795.686} C_VEL
LIN {X 0,Y 175.988,Z 240.039,A -85,B 0,C 180,E1 -24797.029,E2 -24797.029} C_VEL
LIN {X 0,Y 170.762,Z 229.668,A -85,B 0,C 180,E1 -24799.621,E2 -24799.621} C_VEL
LIN {X 0,Y 165.142,Z 220.019,A -85,B 0,C 180,E1 -24802.667,E2 -24802.667} C_VEL
LIN {X 0,Y 159.524,Z 211.312,A -85,B 0,C 180,E1 -24806.111,E2 -24806.111} C_VEL
LIN {X 0,Y 156.062,Z 206.508,A -85,B 0,C 180,E1 -24808.485,E2 -24808.485} C_VEL
LIN {X 0,Y 153.493,Z 202.877,A -85,B 0,C 180,E1 -24810.439,E2 -24810.439} C_VEL
LIN {X 0,Y 150.766,Z 199.368,A -85,B 0,C 180,E1 -24812.698,E2 -24812.698} C_VEL
LIN {X 0,Y 150.045,Z 198.308,A -85,B 0,C 180,E1 -24813.353,E2 -24813.353} C_VEL
LIN {X 0,Y 147.335,Z 195.48,A -85,B 0,C 180,E1 -24815.893,E2 -24815.893} C_VEL
LIN {X 0,Y 146.044,Z 193.146,A -85,B 0,C 180,E1 -24817.357,E2 -24817.357} C_VEL
LIN {X 0,Y 143.448,Z 191.148,A -85,B 0,C 180,E1 -24820.316,E2 -24820.316} C_VEL
LIN {X 0,Y 141.844,Z 188.376,A -85,B 0,C 180,E1 -24822.705,E2 -24822.705} C_VEL
LIN {X 0,Y 141.443,Z 187.488,A -85,B 0,C 180,E1 -24823.399,E2 -24823.399} C_VEL
LIN {X 0,Y 138.679,Z 185.837,A -85,B 0,C 180,E1 -24828.304,E2 -24828.304} C_VEL
LIN {X 0,Y 136.676,Z 181.87,A -85,B 0,C 180,E1 -24836.13,E2 -24836.13} C_VEL
LIN {X 0,Y 136.718,Z 181.456,A -85,B 0,C 180,E1 -24837.053,E2 -24837.053} C_VEL
LIN {X 0,Y 137.111,Z 181.375,A -85,B 0,C 180,E1 -24840,E2 -24840} C_VEL
LIN {X 0,Y 136.696,Z 181.605,A -85,B 0,C 180,E1 -24843.316,E2 -24843.316} C_VEL
LIN {X 0,Y 137.078,Z 183.512,A -85,B 0,C 180,E1 -24846.255,E2 -24846.255} C_VEL
LIN {X 0,Y 140.373,Z 187.102,A -85,B 0,C 180,E1 -24854.497,E2 -24854.497} C_VEL
LIN {X 0,Y 141.608,Z 187.7,A -85,B 0,C 180,E1 -24856.396,E2 -24856.396} C_VEL
LIN {X 0,Y 143.009,Z 190.605,A -85,B 0,C 180,E1 -24858.629,E2 -24858.629} C_VEL
LIN {X 0,Y 145.694,Z 193.009,A -85,B 0,C 180,E1 -24861.82,E2 -24861.82} C_VEL
LIN {X 0,Y 146.329,Z 193.728,A -85,B 0,C 180,E1 -24862.515,E2 -24862.515} C_VEL
LIN {X 0,Y 148.362,Z 196.849,A -85,B 0,C 180,E1 -24864.674,E2 -24864.674} C_VEL
LIN {X 0,Y 150.515,Z 198.96,A -85,B 0,C 180,E1 -24866.604,E2 -24866.604} C_VEL
LIN {X 0,Y 153.127,Z 202.484,A -85,B 0,C 180,E1 -24868.81,E2 -24868.81} C_VEL
LIN {X 0,Y 154.548,Z 204.411,A -85,B 0,C 180,E1 -24869.92,E2 -24869.92} C_VEL
LIN {X 0,Y 157.437,Z 208.364,A -85,B 0,C 180,E1 -24872.016,E2 -24872.016} C_VEL
LIN {X 0,Y 162.577,Z 217.574,A -85,B 0,C 180,E1 -24875.471,E2 -24875.471} C_VEL
LIN {X 0,Y 167.723,Z 228.081,A -85,B 0,C 180,E1 -24878.558,E2 -24878.558} C_VEL
LIN {X 0,Y 171.762,Z 237.532,A -85,B 0,C 180,E1 -24880.798,E2 -24880.798} C_VEL
LIN {X 0,Y 175.415,Z 247.656,A -85,B 0,C 180,E1 -24882.75,E2 -24882.75} C_VEL
LIN {X 0,Y 174.919,Z 257.762,A -85,B 0,C 180,E1 -24883.17,E2 -24883.17} C_VEL
LIN {X 0,Y 172.673,Z 288.253,A -85,B 0,C 180,E1 -24884.284,E2 -24884.284} C_VEL
LIN {X 0,Y 170.692,Z 301.723,A -85,B 0,C 180,E1 -24885.139,E2 -24885.139} C_VEL
LIN {X 0,Y 167.875,Z 314.284,A -85,B 0,C 180,E1 -24886.308,E2 -24886.308} C_VEL
LIN {X 0,Y 164.593,Z 325.355,A -85,B 0,C 180,E1 -24887.738,E2 -24887.738} C_VEL
LIN {X 0,Y 160.459,Z 336.909,A -85,B 0,C 180,E1 -24889.755,E2 -24889.755} C_VEL
LIN {X 0,Y 156.16,Z 347.323,A -85,B 0,C 180,E1 -24892.178,E2 -24892.178} C_VEL
LIN {X 0,Y 152.118,Z 355.837,A -85,B 0,C 180,E1 -24894.723,E2 -24894.723} C_VEL
LIN {X 0,Y 148.102,Z 363.7,A -85,B 0,C 180,E1 -24897.733,E2 -24897.733} C_VEL
LIN {X 0,Y 144.22,Z 370.921,A -85,B 0,C 180,E1 -24901.302,E2 -24901.302} C_VEL
LIN {X 0,Y 141.002,Z 376.662,A -85,B 0,C 180,E1 -24904.932,E2 -24904.932} C_VEL
LIN {X 0,Y 138.009,Z 381.774,A -85,B 0,C 180,E1 -24909.115,E2 -24909.115} C_VEL
LIN {X 0,Y 135.737,Z 385.75,A -85,B 0,C 180,E1 -24913.453,E2 -24913.453} C_VEL
LIN {X 0,Y 134.346,Z 388.698,A -85,B 0,C 180,E1 -24917.92,E2 -24917.92} C_VEL
LIN {X 0,Y 133.462,Z 391.109,A -85,B 0,C 180,E1 -24923.953,E2 -24923.953} C_VEL
LIN {X 0,Y 133.482,Z 391.729,A -85,B 0,C 180,E1 -24926.98,E2 -24926.98} C_VEL
LIN {X 0,Y 133.541,Z 391.912,A -85,B 0,C 180,E1 -24930.676,E2 -24930.676} C_VEL
LIN {X 0,Y 133.534,Z 391.086,A -85,B 0,C 180,E1 -24936.041,E2 -24936.041} C_VEL
LIN {X 0,Y 133.902,Z 389.708,A -85,B 0,C 180,E1 -24939.832,E2 -24939.832} C_VEL
LIN {X 0,Y 133.721,Z 388.527,A -85,B 0,C 180,E1 -24942.304,E2 -24942.304} C_VEL
LIN {X 0,Y 132.121,Z 385.972,A -85,B 0,C 180,E1 -24946.386,E2 -24946.386} C_VEL
LIN {X 0,Y 131.142,Z 382.826,A -85,B 0,C 180,E1 -24950.459,E2 -24950.459} C_VEL
LIN {X 0,Y 131.915,Z 380.527,A -85,B 0,C 180,E1 -24952.806,E2 -24952.806} C_VEL
LIN {X 0,Y 135.843,Z 374.254,A -85,B 0,C 180,E1 -24957.748,E2 -24957.748} C_VEL
LIN {X 0,Y 139.871,Z 367.321,A -85,B 0,C 180,E1 -24961.84,E2 -24961.84} C_VEL
LIN {X 0,Y 143.754,Z 360.248,A -85,B 0,C 180,E1 -24965.059,E2 -24965.059} C_VEL
LIN {X 0,Y 148.167,Z 351.729,A -85,B 0,C 180,E1 -24968.068,E2 -24968.068} C_VEL
LIN {X 0,Y 153.054,Z 341.212,A -85,B 0,C 180,E1 -24970.867,E2 -24970.867} C_VEL
LIN {X 0,Y 157.196,Z 330.804,A -85,B 0,C 180,E1 -24972.982,E2 -24972.982} C_VEL
LIN {X 0,Y 161.059,Z 319.387,A -85,B 0,C 180,E1 -24974.716,E2 -24974.716} C_VEL
LIN {X 0,Y 164.212,Z 307.613,A -85,B 0,C 180,E1 -24976.014,E2 -24976.014} C_VEL
LIN {X 0,Y 166.779,Z 294.083,A -85,B 0,C 180,E1 -24977.059,E2 -24977.059} C_VEL
LIN {X 0,Y 168.165,Z 281.468,A -85,B 0,C 180,E1 -24977.694,E2 -24977.694} C_VEL
LIN {X 0,Y 170.407,Z 249.75,A -85,B 0,C 180,E1 -24978.824,E2 -24978.824} C_VEL
LIN {X 0,Y 165.836,Z 237.19,A -85,B 0,C 180,E1 -24981.487,E2 -24981.487} C_VEL
LIN {X 0,Y 160.373,Z 225.122,A -85,B 0,C 180,E1 -24984.888,E2 -24984.888} C_VEL
LIN {X 0,Y 155.875,Z 216.48,A -85,B 0,C 180,E1 -24988.01,E2 -24988.01} C_VEL
LIN {X 0,Y 153.539,Z 212.583,A -85,B 0,C 180,E1 -24989.768,E2 -24989.768} C_VEL
LIN {X 0,Y 150.727,Z 208.657,A -85,B 0,C 180,E1 -24992.018,E2 -24992.018} C_VEL
LIN {X 0,Y 147.787,Z 204.605,A -85,B 0,C 180,E1 -24994.66,E2 -24994.66} C_VEL
LIN {X 0,Y 144.91,Z 201.131,A -85,B 0,C 180,E1 -24997.578,E2 -24997.578} C_VEL
LIN {X 0,Y 144.072,Z 199.731,A -85,B 0,C 180,E1 -24998.573,E2 -24998.573} C_VEL
LIN {X 0,Y 141.474,Z 197.281,A -85,B 0,C 180,E1 -25001.771,E2 -25001.771} C_VEL
LIN {X 0,Y 139.899,Z 194.35,A -85,B 0,C 180,E1 -25004.335,E2 -25004.335} C_VEL
LIN {X 0,Y 137.368,Z 192.515,A -85,B 0,C 180,E1 -25009.058,E2 -25009.058} C_VEL
LIN {X 0,Y 135.648,Z 188.91,A -85,B 0,C 180,E1 -25015.543,E2 -25015.543} C_VEL
LIN {X 0,Y 135.572,Z 188.441,A -85,B 0,C 180,E1 -25016.285,E2 -25016.285} C_VEL
LIN {X 0,Y 135.395,Z 188.42,A -85,B 0,C 180,E1 -25022.976,E2 -25022.976} C_VEL
LIN {X 0,Y 135.625,Z 188.805,A -85,B 0,C 180,E1 -25024.831,E2 -25024.831} C_VEL
LIN {X 0,Y 137.976,Z 193.226,A -85,B 0,C 180,E1 -25032.876,E2 -25032.876} C_VEL
LIN {X 0,Y 140.122,Z 194.546,A -85,B 0,C 180,E1 -25036.575,E2 -25036.575} C_VEL
LIN {X 0,Y 141.629,Z 197.487,A -85,B 0,C 180,E1 -25039.005,E2 -25039.005} C_VEL
LIN {X 0,Y 144.471,Z 200.239,A -85,B 0,C 180,E1 -25042.445,E2 -25042.445} C_VEL
LIN {X 0,Y 146.945,Z 203.83,A -85,B 0,C 180,E1 -25045.117,E2 -25045.117} C_VEL
LIN {X 0,Y 148.465,Z 205.503,A -85,B 0,C 180,E1 -25046.536,E2 -25046.536} C_VEL
LIN {X 0,Y 151.3,Z 209.271,A -85,B 0,C 180,E1 -25049.002,E2 -25049.002} C_VEL
LIN {X 0,Y 155.813,Z 215.996,A -85,B 0,C 180,E1 -25052.472,E2 -25052.472} C_VEL
LIN {X 0,Y 160.2,Z 222.822,A -85,B 0,C 180,E1 -25055.409,E2 -25055.409} C_VEL
LIN {X 0,Y 165.043,Z 230.973,A -85,B 0,C 180,E1 -25058.3,E2 -25058.3} C_VEL
LIN {X 0,Y 170.57,Z 241.806,A -85,B 0,C 180,E1 -25061.301,E2 -25061.301} C_VEL
LIN {X 0,Y 170.895,Z 242.559,A -85,B 0,C 180,E1 -25061.473,E2 -25061.473} C_VEL
LIN {X 0,Y 168.195,Z 279.509,A -85,B 0,C 180,E1 -25062.857,E2 -25062.857} C_VEL
LIN {X 0,Y 166.276,Z 292.612,A -85,B 0,C 180,E1 -25063.708,E2 -25063.708} C_VEL
LIN {X 0,Y 163.709,Z 304.773,A -85,B 0,C 180,E1 -25064.903,E2 -25064.903} C_VEL
LIN {X 0,Y 160.653,Z 316.04,A -85,B 0,C 180,E1 -25066.451,E2 -25066.451} C_VEL
LIN {X 0,Y 156.505,Z 327.655,A -85,B 0,C 180,E1 -25068.522,E2 -25068.522} C_VEL
LIN {X 0,Y 152.153,Z 338.085,A -85,B 0,C 180,E1 -25071.001,E2 -25071.001} C_VEL
LIN {X 0,Y 147.726,Z 347.551,A -85,B 0,C 180,E1 -25073.976,E2 -25073.976} C_VEL
LIN {X 0,Y 143.317,Z 355.825,A -85,B 0,C 180,E1 -25077.358,E2 -25077.358} C_VEL
LIN {X 0,Y 138.906,Z 363.217,A -85,B 0,C 180,E1 -25081.274,E2 -25081.274} C_VEL
LIN {X 0,Y 135.109,Z 369.147,A -85,B 0,C 180,E1 -25085.411,E2 -25085.411} C_VEL
LIN {X 0,Y 132.038,Z 373.827,A -85,B 0,C 180,E1 -25089.761,E2 -25089.761} C_VEL
LIN {X 0,Y 129.663,Z 377.404,A -85,B 0,C 180,E1 -25094.278,E2 -25094.278} C_VEL
LIN {X 0,Y 128.474,Z 379.25,A -85,B 0,C 180,E1 -25097.362,E2 -25097.362} C_VEL
LIN {X 0,Y 127.633,Z 380.632,A -85,B 0,C 180,E1 -25100.493,E2 -25100.493} C_VEL
LIN {X 0,Y 126.7,Z 382.22,A -85,B 0,C 180,E1 -25106.822,E2 -25106.822} C_VEL
LIN {X 0,Y 126.633,Z 382.444,A -85,B 0,C 180,E1 -25110.002,E2 -25110.002} C_VEL
LIN {X 0,Y 126.7,Z 382.25,A -85,B 0,C 180,E1 -25113.181,E2 -25113.181} C_VEL
LIN {X 0,Y 127.633,Z 380.7,A -85,B 0,C 180,E1 -25119.51,E2 -25119.51} C_VEL
LIN {X 0,Y 128.461,Z 379.347,A -85,B 0,C 180,E1 -25122.642,E2 -25122.642} C_VEL
LIN {X 0,Y 130.331,Z 376.484,A -85,B 0,C 180,E1 -25127.254,E2 -25127.254} C_VEL
LIN {X 0,Y 132.953,Z 372.596,A -85,B 0,C 180,E1 -25131.719,E2 -25131.719} C_VEL
LIN {X 0,Y 136.226,Z 367.58,A -85,B 0,C 180,E1 -25136.011,E2 -25136.011} C_VEL
LIN {X 0,Y 140.244,Z 361.254,A -85,B 0,C 180,E1 -25140.076,E2 -25140.076} C_VEL
LIN {X 0,Y 144.832,Z 353.339,A -85,B 0,C 180,E1 -25143.922,E2 -25143.922} C_VEL
LIN {X 0,Y 149.819,Z 343.499,A -85,B 0,C 180,E1 -25147.578,E2 -25147.578} C_VEL
LIN {X 0,Y 154.478,Z 333.151,A -85,B 0,C 180,E1 -25150.415,E2 -25150.415} C_VEL
LIN {X 0,Y 158.947,Z 321.479,A -85,B 0,C 180,E1 -25152.831,E2 -25152.831} C_VEL
LIN {X 0,Y 162.579,Z 309.818,A -85,B 0,C 180,E1 -25154.626,E2 -25154.626} C_VEL
LIN {X 0,Y 165.545,Z 297.679,A -85,B 0,C 180,E1 -25155.978,E2 -25155.978} C_VEL
LIN {X 0,Y 167.804,Z 284.449,A -85,B 0,C 180,E1 -25157.018,E2 -25157.018} C_VEL
LIN {X 0,Y 169.232,Z 270.762,A -85,B 0,C 180,E1 -25157.626,E2 -25157.626} C_VEL
LIN {X 0,Y 171.056,Z 242.647,A -85,B 0,C 180,E1 -25158.685,E2 -25158.685} C_VEL
LIN {X 0,Y 165.888,Z 232.425,A -85,B 0,C 180,E1 -25161.471,E2 -25161.471} C_VEL
LIN {X 0,Y 160.68,Z 223.44,A -85,B 0,C 180,E1 -25164.565,E2 -25164.565} C_VEL
LIN {X 0,Y 156.116,Z 216.32,A -85,B 0,C 180,E1 -25167.612,E2 -25167.612} C_VEL
LIN {X 0,Y 153.196,Z 212.056,A -85,B 0,C 180,E1 -25169.783,E2 -25169.783} C_VEL
LIN {X 0,Y 151.131,Z 209.059,A -85,B 0,C 180,E1 -25171.462,E2 -25171.462} C_VEL
LIN {X 0,Y 148.278,Z 205.051,A -85,B 0,C 180,E1 -25174.017,E2 -25174.017} C_VEL
LIN {X 0,Y 145.184,Z 201.492,A -85,B 0,C 180,E1 -25177.122,E2 -25177.122} C_VEL
LIN {X 0,Y 144.16,Z 199.735,A -85,B 0,C 180,E1 -25178.351,E2 -25178.351} C_VEL
LIN {X 0,Y 141.589,Z 197.392,A -85,B 0,C 180,E1 -25181.552,E2 -25181.552} C_VEL
LIN {X 0,Y 140.13,Z 194.502,A -85,B 0,C 180,E1 -25183.987,E2 -25183.987} C_VEL
LIN {X 0,Y 137.142,Z 192.2,A -85,B 0,C 180,E1 -25189.947,E2 -25189.947} C_VEL
LIN {X 0,Y 135.739,Z 188.697,A -85,B 0,C 180,E1 -25196.846,E2 -25196.846} C_VEL
LIN {X 0,Y 135.66,Z 188.399,A -85,B 0,C 180,E1 -25201.484,E2 -25201.484} C_VEL
LIN {X 0,Y 135.763,Z 188.788,A -85,B 0,C 180,E1 -25202.967,E2 -25202.967} C_VEL
LIN {X 0,Y 136.57,Z 191.311,A -85,B 0,C 180,E1 -25207.763,E2 -25207.763} C_VEL
LIN {X 0,Y 139.32,Z 194.093,A -85,B 0,C 180,E1 -25214.236,E2 -25214.236} C_VEL
LIN {X 0,Y 140.172,Z 194.661,A -85,B 0,C 180,E1 -25215.634,E2 -25215.634} C_VEL
LIN {X 0,Y 142.138,Z 198.092,A -85,B 0,C 180,E1 -25218.747,E2 -25218.747} C_VEL
LIN {X 0,Y 144.413,Z 200.139,A -85,B 0,C 180,E1 -25221.488,E2 -25221.488} C_VEL
LIN {X 0,Y 146.696,Z 203.573,A -85,B 0,C 180,E1 -25224.03,E2 -25224.03} C_VEL
LIN {X 0,Y 148.468,Z 205.446,A -85,B 0,C 180,E1 -25225.709,E2 -25225.709} C_VEL
LIN {X 0,Y 151.99,Z 210.326,A -85,B 0,C 180,E1 -25228.786,E2 -25228.786} C_VEL
LIN {X 0,Y 154.77,Z 214.317,A -85,B 0,C 180,E1 -25230.942,E2 -25230.942} C_VEL
LIN {X 0,Y 159.633,Z 223.493,A -85,B 0,C 180,E1 -25234.434,E2 -25234.434} C_VEL
LIN {X 0,Y 164.023,Z 232.851,A -85,B 0,C 180,E1 -25237.258,E2 -25237.258} C_VEL
LIN {X 0,Y 167.674,Z 241.689,A -85,B 0,C 180,E1 -25239.44,E2 -25239.44} C_VEL
LIN {X 0,Y 170.61,Z 249.968,A -85,B 0,C 180,E1 -25241.133,E2 -25241.133} C_VEL
LIN {X 0,Y 167.805,Z 288.049,A -85,B 0,C 180,E1 -25242.557,E2 -25242.557} C_VEL
LIN {X 0,Y 165.685,Z 301.738,A -85,B 0,C 180,E1 -25243.427,E2 -25243.427} C_VEL
LIN {X 0,Y 162.828,Z 314.031,A -85,B 0,C 180,E1 -25244.587,E2 -25244.587} C_VEL
LIN {X 0,Y 159.411,Z 325.101,A -85,B 0,C 180,E1 -25246.022,E2 -25246.022} C_VEL
LIN {X 0,Y 155.107,Z 336.654,A -85,B 0,C 180,E1 -25248.061,E2 -25248.061} C_VEL
LIN {X 0,Y 150.613,Z 347.067,A -85,B 0,C 180,E1 -25250.521,E2 -25250.521} C_VEL
LIN {X 0,Y 146.353,Z 355.579,A -85,B 0,C 180,E1 -25253.11,E2 -25253.11} C_VEL
LIN {X 0,Y 141.347,Z 364.817,A -85,B 0,C 180,E1 -25256.842,E2 -25256.842} C_VEL
LIN {X 0,Y 136.891,Z 372.492,A -85,B 0,C 180,E1 -25260.987,E2 -25260.987} C_VEL
LIN {X 0,Y 133.396,Z 378.227,A -85,B 0,C 180,E1 -25265.071,E2 -25265.071} C_VEL
LIN {X 0,Y 130.463,Z 382.952,A -85,B 0,C 180,E1 -25269.502,E2 -25269.502} C_VEL
LIN {X 0,Y 128.322,Z 386.569,A -85,B 0,C 180,E1 -25274.106,E2 -25274.106} C_VEL
LIN {X 0,Y 127.382,Z 388.439,A -85,B 0,C 180,E1 -25277.249,E2 -25277.249} C_VEL
LIN {X 0,Y 126.401,Z 390.85,A -85,B 0,C 180,E1 -25283.614,E2 -25283.614} C_VEL
LIN {X 0,Y 126.383,Z 391.469,A -85,B 0,C 180,E1 -25286.811,E2 -25286.811} C_VEL
LIN {X 0,Y 126.504,Z 391.687,A -85,B 0,C 180,E1 -25289.998,E2 -25289.998} C_VEL
LIN {X 0,Y 126.378,Z 391.453,A -85,B 0,C 180,E1 -25293.186,E2 -25293.186} C_VEL
LIN {X 0,Y 126.455,Z 390.826,A -85,B 0,C 180,E1 -25296.38,E2 -25296.38} C_VEL
LIN {X 0,Y 126.829,Z 389.604,A -85,B 0,C 180,E1 -25300.03,E2 -25300.03} C_VEL
LIN {X 0,Y 127.384,Z 388.386,A -85,B 0,C 180,E1 -25302.747,E2 -25302.747} C_VEL
LIN {X 0,Y 128.901,Z 385.415,A -85,B 0,C 180,E1 -25307.448,E2 -25307.448} C_VEL
LIN {X 0,Y 131.915,Z 380.527,A -85,B 0,C 180,E1 -25312.806,E2 -25312.806} C_VEL
LIN {X 0,Y 132.873,Z 378.029,A -85,B 0,C 180,E1 -25315.082,E2 -25315.082} C_VEL
LIN {X 0,Y 133.051,Z 373.523,A -85,B 0,C 180,E1 -25318.895,E2 -25318.895} C_VEL
LIN {X 0,Y 133.593,Z 368.442,A -85,B 0,C 180,E1 -25322.555,E2 -25322.555} C_VEL
LIN {X 0,Y 135.059,Z 364.976,A -85,B 0,C 180,E1 -25324.506,E2 -25324.506} C_VEL
LIN {X 0,Y 139.78,Z 356.753,A -85,B 0,C 180,E1 -25328.016,E2 -25328.016} C_VEL
LIN {X 0,Y 144.66,Z 347.55,A -85,B 0,C 180,E1 -25330.983,E2 -25330.983} C_VEL
LIN {X 0,Y 149.321,Z 337.312,A -85,B 0,C 180,E1 -25333.497,E2 -25333.497} C_VEL
LIN {X 0,Y 153.787,Z 325.966,A -85,B 0,C 180,E1 -25335.563,E2 -25335.563} C_VEL
LIN {X 0,Y 157.599,Z 314.186,A -85,B 0,C 180,E1 -25337.137,E2 -25337.137} C_VEL
LIN {X 0,Y 160.629,Z 301.664,A -85,B 0,C 180,E1 -25338.34,E2 -25338.34} C_VEL
LIN {X 0,Y 162.793,Z 288.386,A -85,B 0,C 180,E1 -25339.195,E2 -25339.195} C_VEL
LIN {X 0,Y 164.486,Z 268.475,A -85,B 0,C 180,E1 -25339.962,E2 -25339.962} C_VEL
LIN {X 0,Y 165.631,Z 252,A -85,B 0,C 180,E1 -25340.58,E2 -25340.58} C_VEL
LIN {X 0,Y 161.777,Z 241.11,A -85,B 0,C 180,E1 -25343.029,E2 -25343.029} C_VEL
LIN {X 0,Y 156.831,Z 229.77,A -85,B 0,C 180,E1 -25346.376,E2 -25346.376} C_VEL
LIN {X 0,Y 152.611,Z 221.337,A -85,B 0,C 180,E1 -25349.565,E2 -25349.565} C_VEL
LIN {X 0,Y 150.95,Z 218.508,A -85,B 0,C 180,E1 -25350.911,E2 -25350.911} C_VEL
LIN {X 0,Y 148.425,Z 214.774,A -85,B 0,C 180,E1 -25353.077,E2 -25353.077} C_VEL
LIN {X 0,Y 145.601,Z 210.866,A -85,B 0,C 180,E1 -25355.777,E2 -25355.777} C_VEL
LIN {X 0,Y 142.727,Z 206.919,A -85,B 0,C 180,E1 -25358.975,E2 -25358.975} C_VEL
LIN {X 0,Y 139.377,Z 202.964,A -85,B 0,C 180,E1 -25363.523,E2 -25363.523} C_VEL
LIN {X 0,Y 138.608,Z 201.256,A -85,B 0,C 180,E1 -25364.938,E2 -25364.938} C_VEL
LIN {X 0,Y 135.986,Z 199.071,A -85,B 0,C 180,E1 -25370.32,E2 -25370.32} C_VEL
LIN {X 0,Y 134.663,Z 195.612,A -85,B 0,C 180,E1 -25376.447,E2 -25376.447} C_VEL
LIN {X 0,Y 134.402,Z 195.301,A -85,B 0,C 180,E1 -25380,E2 -25380} C_VEL
LIN {X 0,Y 134.672,Z 195.791,A -85,B 0,C 180,E1 -25384.302,E2 -25384.302} C_VEL
LIN {X 0,Y 136.949,Z 200.223,A -85,B 0,C 180,E1 -25392.598,E2 -25392.598} C_VEL
LIN {X 0,Y 138.739,Z 201.516,A -85,B 0,C 180,E1 -25395.866,E2 -25395.866} C_VEL
LIN {X 0,Y 140.637,Z 204.81,A -85,B 0,C 180,E1 -25398.955,E2 -25398.955} C_VEL
LIN {X 0,Y 142.727,Z 206.876,A -85,B 0,C 180,E1 -25401.578,E2 -25401.578} C_VEL
LIN {X 0,Y 145.288,Z 210.517,A -85,B 0,C 180,E1 -25404.469,E2 -25404.469} C_VEL
LIN {X 0,Y 146.503,Z 212.089,A -85,B 0,C 180,E1 -25405.682,E2 -25405.682} C_VEL
LIN {X 0,Y 149.674,Z 216.592,A -85,B 0,C 180,E1 -25408.579,E2 -25408.579} C_VEL
LIN {X 0,Y 152.819,Z 221.369,A -85,B 0,C 180,E1 -25411.128,E2 -25411.128} C_VEL
LIN {X 0,Y 157.165,Z 228.366,A -85,B 0,C 180,E1 -25414.251,E2 -25414.251} C_VEL
LIN {X 0,Y 161.858,Z 236.686,A -85,B 0,C 180,E1 -25417.249,E2 -25417.249} C_VEL
LIN {X 0,Y 166.084,Z 245.112,A -85,B 0,C 180,E1 -25419.709,E2 -25419.709} C_VEL
LIN {X 0,Y 163.95,Z 274.56,A -85,B 0,C 180,E1 -25420.796,E2 -25420.796} C_VEL
LIN {X 0,Y 162.239,Z 288.484,A -85,B 0,C 180,E1 -25421.553,E2 -25421.553} C_VEL
LIN {X 0,Y 159.904,Z 300.515,A -85,B 0,C 180,E1 -25422.595,E2 -25422.595} C_VEL
LIN {X 0,Y 156.63,Z 312.82,A -85,B 0,C 180,E1 -25424.12,E2 -25424.12} C_VEL
LIN {X 0,Y 152.863,Z 323.876,A -85,B 0,C 180,E1 -25425.945,E2 -25425.945} C_VEL
LIN {X 0,Y 148.172,Z 335.149,A -85,B 0,C 180,E1 -25428.394,E2 -25428.394} C_VEL
LIN {X 0,Y 143.361,Z 345.175,A -85,B 0,C 180,E1 -25431.36,E2 -25431.36} C_VEL
LIN {X 0,Y 139.079,Z 353.227,A -85,B 0,C 180,E1 -25434.473,E2 -25434.473} C_VEL
LIN {X 0,Y 134.222,Z 361.205,A -85,B 0,C 180,E1 -25438.428,E2 -25438.428} C_VEL
LIN {X 0,Y 129.943,Z 367.605,A -85,B 0,C 180,E1 -25442.633,E2 -25442.633} C_VEL
LIN {X 0,Y 126.435,Z 372.674,A -85,B 0,C 180,E1 -25447.104,E2 -25447.104} C_VEL
LIN {X 0,Y 123.619,Z 376.608,A -85,B 0,C 180,E1 -25451.781,E2 -25451.781} C_VEL
LIN {X 0,Y 121.572,Z 379.509,A -85,B 0,C 180,E1 -25456.632,E2 -25456.632} C_VEL
LIN {X 0,Y 120.627,Z 380.892,A -85,B 0,C 180,E1 -25459.936,E2 -25459.936} C_VEL
LIN {X 0,Y 119.625,Z 382.479,A -85,B 0,C 180,E1 -25466.634,E2 -25466.634} C_VEL
LIN {X 0,Y 119.528,Z 382.638,A -85,B 0,C 180,E1 -25471.685,E2 -25471.685} C_VEL
LIN {X 0,Y 119.988,Z 381.924,A -85,B 0,C 180,E1 -25476.729,E2 -25476.729} C_VEL
LIN {X 0,Y 120.626,Z 380.959,A -85,B 0,C 180,E1 -25480.068,E2 -25480.068} C_VEL
LIN {X 0,Y 121.537,Z 379.606,A -85,B 0,C 180,E1 -25483.375,E2 -25483.375} C_VEL
LIN {X 0,Y 123.575,Z 376.742,A -85,B 0,C 180,E1 -25488.229,E2 -25488.229} C_VEL
LIN {X 0,Y 126.396,Z 372.854,A -85,B 0,C 180,E1 -25492.908,E2 -25492.908} C_VEL
LIN {X 0,Y 129.889,Z 367.837,A -85,B 0,C 180,E1 -25497.383,E2 -25497.383} C_VEL
LIN {X 0,Y 134.158,Z 361.51,A -85,B 0,C 180,E1 -25501.593,E2 -25501.593} C_VEL
LIN {X 0,Y 138.889,Z 353.786,A -85,B 0,C 180,E1 -25505.472,E2 -25505.472} C_VEL
LIN {X 0,Y 143.275,Z 345.707,A -85,B 0,C 180,E1 -25508.624,E2 -25508.624} C_VEL
LIN {X 0,Y 148.122,Z 335.681,A -85,B 0,C 180,E1 -25511.627,E2 -25511.627} C_VEL
LIN {X 0,Y 152.791,Z 324.575,A -85,B 0,C 180,E1 -25514.085,E2 -25514.085} C_VEL
LIN {X 0,Y 156.552,Z 313.687,A -85,B 0,C 180,E1 -25515.914,E2 -25515.914} C_VEL
LIN {X 0,Y 159.568,Z 302.773,A -85,B 0,C 180,E1 -25517.307,E2 -25517.307} C_VEL
LIN {X 0,Y 162.274,Z 289.806,A -85,B 0,C 180,E1 -25518.492,E2 -25518.492} C_VEL
LIN {X 0,Y 163.951,Z 277.282,A -85,B 0,C 180,E1 -25519.224,E2 -25519.224} C_VEL
LIN {X 0,Y 166.233,Z 246.773,A -85,B 0,C 180,E1 -25520.354,E2 -25520.354} C_VEL
LIN {X 0,Y 166.14,Z 245.062,A -85,B 0,C 180,E1 -25520.507,E2 -25520.507} C_VEL
